Fanuc TP program (LS listing): FM152932.ls

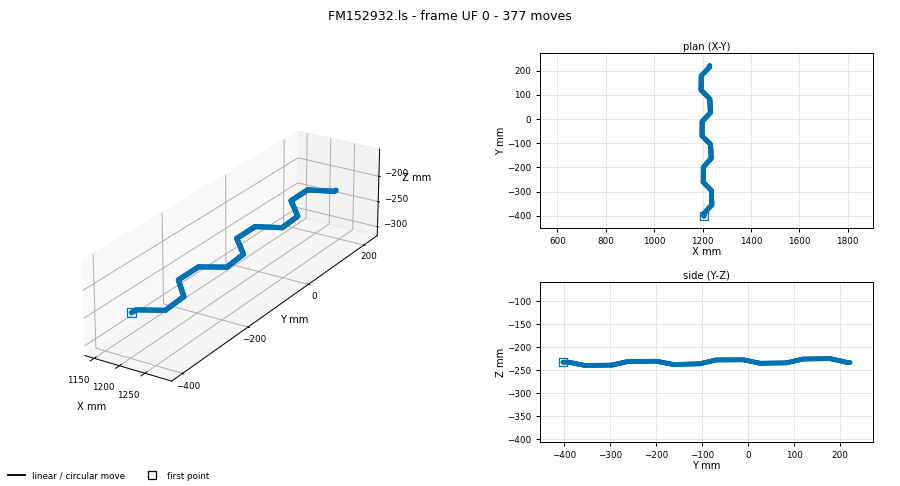
[picture p0: tool path of FM152932.ls in frame UF 0, 377 of 377 moves have a stored position in this frame; points joined in program order, loops and branches not executed]
/PROG  FM152932
/ATTR
OWNER		= MNEDITOR;
COMMENT		= "Auto FANUC move";
PROG_SIZE	= 0;
CREATE		= DATE 26-05-06  TIME 15:29:32;
MODIFIED	= DATE 26-05-06  TIME 15:29:32;
FILE_NAME	= ;
VERSION		= 0;
LINE_COUNT	= 382;
MEMORY_SIZE	= 0;
PROTECT		= READ_WRITE;
TCD:  STACK_SIZE	= 0,
      TASK_PRIORITY	= 50,
      TIME_SLICE	= 0,
      BUSY_LAMP_OFF	= 0,
      ABORT_REQUEST	= 0,
      PAUSE_REQUEST	= 0;
DEFAULT_GROUP	= 1,*,*,*,*;
CONTROL_CODE	= 00000000 00000000;
/MN
   1:  UFRAME_NUM=0 ;
   2:  UTOOL_NUM=1 ;
   3:  R[93]=10 ;
   4:  L P[1] 7mm/sec FINE ;
   5:  L P[2] 7mm/sec CNT50 ;
   6:  L P[3] 7mm/sec CNT50 ;
   7:  L P[4] 7mm/sec CNT50 ;
   8:  L P[5] 7mm/sec CNT50 ;
   9:  L P[6] 7mm/sec CNT50 ;
  10:  L P[7] 7mm/sec CNT50 ;
  11:  L P[8] 7mm/sec CNT50 ;
  12:  L P[9] 7mm/sec CNT50 ;
  13:  L P[10] 7mm/sec CNT50 ;
  14:  L P[11] 7mm/sec CNT50 ;
  15:  L P[12] 7mm/sec CNT50 ;
  16:  L P[13] 7mm/sec CNT50 ;
  17:  L P[14] 7mm/sec CNT50 ;
  18:  L P[15] 7mm/sec CNT50 ;
  19:  L P[16] 7mm/sec CNT50 ;
  20:  L P[17] 7mm/sec CNT50 ;
  21:  L P[18] 7mm/sec CNT50 ;
  22:  L P[19] 7mm/sec CNT50 ;
  23:  L P[20] 7mm/sec CNT50 ;
  24:  L P[21] 7mm/sec CNT50 ;
  25:  L P[22] 7mm/sec CNT50 ;
  26:  L P[23] 7mm/sec CNT50 ;
  27:  L P[24] 7mm/sec CNT50 ;
  28:  L P[25] 7mm/sec CNT50 ;
  29:  L P[26] 7mm/sec CNT50 ;
  30:  L P[27] 7mm/sec CNT50 ;
  31:  L P[28] 7mm/sec CNT50 ;
  32:  L P[29] 7mm/sec CNT50 ;
  33:  L P[30] 7mm/sec CNT50 ;
  34:  L P[31] 7mm/sec CNT50 ;
  35:  L P[32] 7mm/sec CNT50 ;
  36:  L P[33] 7mm/sec CNT50 ;
  37:  L P[34] 7mm/sec CNT50 ;
  38:  L P[35] 7mm/sec CNT50 ;
  39:  L P[36] 7mm/sec CNT50 ;
  40:  L P[37] 7mm/sec CNT50 ;
  41:  L P[38] 7mm/sec CNT50 ;
  42:  L P[39] 7mm/sec CNT50 ;
  43:  L P[40] 7mm/sec CNT50 ;
  44:  L P[41] 7mm/sec CNT50 ;
  45:  L P[42] 7mm/sec CNT50 ;
  46:  L P[43] 7mm/sec CNT50 ;
  47:  L P[44] 7mm/sec CNT50 ;
  48:  L P[45] 7mm/sec CNT50 ;
  49:  L P[46] 7mm/sec CNT50 ;
  50:  L P[47] 7mm/sec CNT50 ;
  51:  L P[48] 7mm/sec CNT50 ;
  52:  L P[49] 7mm/sec CNT50 ;
  53:  L P[50] 7mm/sec CNT50 ;
  54:  L P[51] 7mm/sec CNT50 ;
  55:  L P[52] 7mm/sec CNT50 ;
  56:  L P[53] 7mm/sec CNT50 ;
  57:  L P[54] 7mm/sec CNT50 ;
  58:  L P[55] 7mm/sec CNT50 ;
  59:  L P[56] 7mm/sec CNT50 ;
  60:  L P[57] 7mm/sec CNT50 ;
  61:  L P[58] 7mm/sec CNT50 ;
  62:  L P[59] 7mm/sec CNT50 ;
  63:  L P[60] 7mm/sec CNT50 ;
  64:  L P[61] 7mm/sec CNT50 ;
  65:  L P[62] 7mm/sec CNT50 ;
  66:  L P[63] 7mm/sec CNT50 ;
  67:  L P[64] 7mm/sec CNT50 ;
  68:  L P[65] 7mm/sec CNT50 ;
  69:  L P[66] 7mm/sec CNT50 ;
  70:  L P[67] 7mm/sec CNT50 ;
  71:  L P[68] 7mm/sec CNT50 ;
  72:  L P[69] 7mm/sec CNT50 ;
  73:  L P[70] 7mm/sec CNT50 ;
  74:  L P[71] 7mm/sec CNT50 ;
  75:  L P[72] 7mm/sec CNT50 ;
  76:  L P[73] 7mm/sec CNT50 ;
  77:  L P[74] 7mm/sec CNT50 ;
  78:  L P[75] 7mm/sec CNT50 ;
  79:  L P[76] 7mm/sec CNT50 ;
  80:  L P[77] 7mm/sec CNT50 ;
  81:  L P[78] 7mm/sec CNT50 ;
  82:  L P[79] 7mm/sec CNT50 ;
  83:  L P[80] 7mm/sec CNT50 ;
  84:  L P[81] 7mm/sec CNT50 ;
  85:  L P[82] 7mm/sec CNT50 ;
  86:  L P[83] 7mm/sec CNT50 ;
  87:  L P[84] 7mm/sec CNT50 ;
  88:  L P[85] 7mm/sec CNT50 ;
  89:  L P[86] 7mm/sec CNT50 ;
  90:  L P[87] 7mm/sec CNT50 ;
  91:  L P[88] 7mm/sec CNT50 ;
  92:  L P[89] 7mm/sec CNT50 ;
  93:  L P[90] 7mm/sec CNT50 ;
  94:  L P[91] 7mm/sec CNT50 ;
  95:  L P[92] 7mm/sec CNT50 ;
  96:  L P[93] 7mm/sec CNT50 ;
  97:  L P[94] 7mm/sec CNT50 ;
  98:  L P[95] 7mm/sec CNT50 ;
  99:  L P[96] 7mm/sec CNT50 ;
 100:  L P[97] 7mm/sec CNT50 ;
 101:  L P[98] 7mm/sec CNT50 ;
 102:  L P[99] 7mm/sec CNT50 ;
 103:  L P[100] 7mm/sec CNT50 ;
 104:  L P[101] 7mm/sec CNT50 ;
 105:  L P[102] 7mm/sec CNT50 ;
 106:  L P[103] 7mm/sec CNT50 ;
 107:  L P[104] 7mm/sec CNT50 ;
 108:  L P[105] 7mm/sec CNT50 ;
 109:  L P[106] 7mm/sec CNT50 ;
 110:  L P[107] 7mm/sec CNT50 ;
 111:  L P[108] 7mm/sec CNT50 ;
 112:  L P[109] 7mm/sec CNT50 ;
 113:  L P[110] 7mm/sec CNT50 ;
 114:  L P[111] 7mm/sec CNT50 ;
 115:  L P[112] 7mm/sec CNT50 ;
 116:  L P[113] 7mm/sec CNT50 ;
 117:  L P[114] 7mm/sec CNT50 ;
 118:  L P[115] 7mm/sec CNT50 ;
 119:  L P[116] 7mm/sec CNT50 ;
 120:  L P[117] 7mm/sec CNT50 ;
 121:  L P[118] 7mm/sec CNT50 ;
 122:  L P[119] 7mm/sec CNT50 ;
 123:  L P[120] 7mm/sec CNT50 ;
 124:  L P[121] 7mm/sec CNT50 ;
 125:  L P[122] 7mm/sec CNT50 ;
 126:  L P[123] 7mm/sec CNT50 ;
 127:  L P[124] 7mm/sec CNT50 ;
 128:  L P[125] 7mm/sec CNT50 ;
 129:  L P[126] 7mm/sec CNT50 ;
 130:  L P[127] 7mm/sec CNT50 ;
 131:  L P[128] 7mm/sec CNT50 ;
 132:  L P[129] 7mm/sec CNT50 ;
 133:  L P[130] 7mm/sec CNT50 ;
 134:  L P[131] 7mm/sec CNT50 ;
 135:  L P[132] 7mm/sec CNT50 ;
 136:  L P[133] 7mm/sec CNT50 ;
 137:  L P[134] 7mm/sec CNT50 ;
 138:  L P[135] 7mm/sec CNT50 ;
 139:  L P[136] 7mm/sec CNT50 ;
 140:  L P[137] 7mm/sec CNT50 ;
 141:  L P[138] 7mm/sec CNT50 ;
 142:  L P[139] 7mm/sec CNT50 ;
 143:  L P[140] 7mm/sec CNT50 ;
 144:  L P[141] 7mm/sec CNT50 ;
 145:  L P[142] 7mm/sec CNT50 ;
 146:  L P[143] 7mm/sec CNT50 ;
 147:  L P[144] 7mm/sec CNT50 ;
 148:  L P[145] 7mm/sec CNT50 ;
 149:  L P[146] 7mm/sec CNT50 ;
 150:  L P[147] 7mm/sec CNT50 ;
 151:  L P[148] 7mm/sec CNT50 ;
 152:  L P[149] 7mm/sec CNT50 ;
 153:  L P[150] 7mm/sec CNT50 ;
 154:  L P[151] 7mm/sec CNT50 ;
 155:  L P[152] 7mm/sec CNT50 ;
 156:  L P[153] 7mm/sec CNT50 ;
 157:  L P[154] 7mm/sec CNT50 ;
 158:  L P[155] 7mm/sec CNT50 ;
 159:  L P[156] 7mm/sec CNT50 ;
 160:  L P[157] 7mm/sec CNT50 ;
 161:  L P[158] 7mm/sec CNT50 ;
 162:  L P[159] 7mm/sec CNT50 ;
 163:  L P[160] 7mm/sec CNT50 ;
 164:  L P[161] 7mm/sec CNT50 ;
 165:  L P[162] 7mm/sec CNT50 ;
 166:  L P[163] 7mm/sec CNT50 ;
 167:  L P[164] 7mm/sec CNT50 ;
 168:  L P[165] 7mm/sec CNT50 ;
 169:  L P[166] 7mm/sec CNT50 ;
 170:  L P[167] 7mm/sec CNT50 ;
 171:  L P[168] 7mm/sec CNT50 ;
 172:  L P[169] 7mm/sec CNT50 ;
 173:  L P[170] 7mm/sec CNT50 ;
 174:  L P[171] 7mm/sec CNT50 ;
 175:  L P[172] 7mm/sec CNT50 ;
 176:  L P[173] 7mm/sec CNT50 ;
 177:  L P[174] 7mm/sec CNT50 ;
 178:  L P[175] 7mm/sec CNT50 ;
 179:  L P[176] 7mm/sec CNT50 ;
 180:  L P[177] 7mm/sec CNT50 ;
 181:  L P[178] 7mm/sec CNT50 ;
 182:  L P[179] 7mm/sec CNT50 ;
 183:  L P[180] 7mm/sec CNT50 ;
 184:  L P[181] 7mm/sec CNT50 ;
 185:  L P[182] 7mm/sec CNT50 ;
 186:  L P[183] 7mm/sec CNT50 ;
 187:  L P[184] 7mm/sec CNT50 ;
 188:  L P[185] 7mm/sec CNT50 ;
 189:  L P[186] 7mm/sec CNT50 ;
 190:  L P[187] 7mm/sec CNT50 ;
 191:  L P[188] 7mm/sec CNT50 ;
 192:  L P[189] 7mm/sec CNT50 ;
 193:  L P[190] 7mm/sec CNT50 ;
 194:  L P[191] 7mm/sec CNT50 ;
 195:  L P[192] 7mm/sec CNT50 ;
 196:  L P[193] 7mm/sec CNT50 ;
 197:  L P[194] 7mm/sec CNT50 ;
 198:  L P[195] 7mm/sec CNT50 ;
 199:  L P[196] 7mm/sec CNT50 ;
 200:  L P[197] 7mm/sec CNT50 ;
 201:  L P[198] 7mm/sec CNT50 ;
 202:  L P[199] 7mm/sec CNT50 ;
 203:  L P[200] 7mm/sec CNT50 ;
 204:  L P[201] 7mm/sec CNT50 ;
 205:  L P[202] 7mm/sec CNT50 ;
 206:  L P[203] 7mm/sec CNT50 ;
 207:  L P[204] 7mm/sec CNT50 ;
 208:  L P[205] 7mm/sec CNT50 ;
 209:  L P[206] 7mm/sec CNT50 ;
 210:  L P[207] 7mm/sec CNT50 ;
 211:  L P[208] 7mm/sec CNT50 ;
 212:  L P[209] 7mm/sec CNT50 ;
 213:  L P[210] 7mm/sec CNT50 ;
 214:  L P[211] 7mm/sec CNT50 ;
 215:  L P[212] 7mm/sec CNT50 ;
 216:  L P[213] 7mm/sec CNT50 ;
 217:  L P[214] 7mm/sec CNT50 ;
 218:  L P[215] 7mm/sec CNT50 ;
 219:  L P[216] 7mm/sec CNT50 ;
 220:  L P[217] 7mm/sec CNT50 ;
 221:  L P[218] 7mm/sec CNT50 ;
 222:  L P[219] 7mm/sec CNT50 ;
 223:  L P[220] 7mm/sec CNT50 ;
 224:  L P[221] 7mm/sec CNT50 ;
 225:  L P[222] 7mm/sec CNT50 ;
 226:  L P[223] 7mm/sec CNT50 ;
 227:  L P[224] 7mm/sec CNT50 ;
 228:  L P[225] 7mm/sec CNT50 ;
 229:  L P[226] 7mm/sec CNT50 ;
 230:  L P[227] 7mm/sec CNT50 ;
 231:  L P[228] 7mm/sec CNT50 ;
 232:  L P[229] 7mm/sec CNT50 ;
 233:  L P[230] 7mm/sec CNT50 ;
 234:  L P[231] 7mm/sec CNT50 ;
 235:  L P[232] 7mm/sec CNT50 ;
 236:  L P[233] 7mm/sec CNT50 ;
 237:  L P[234] 7mm/sec CNT50 ;
 238:  L P[235] 7mm/sec CNT50 ;
 239:  L P[236] 7mm/sec CNT50 ;
 240:  L P[237] 7mm/sec CNT50 ;
 241:  L P[238] 7mm/sec CNT50 ;
 242:  L P[239] 7mm/sec CNT50 ;
 243:  L P[240] 7mm/sec CNT50 ;
 244:  L P[241] 7mm/sec CNT50 ;
 245:  L P[242] 7mm/sec CNT50 ;
 246:  L P[243] 7mm/sec CNT50 ;
 247:  L P[244] 7mm/sec CNT50 ;
 248:  L P[245] 7mm/sec CNT50 ;
 249:  L P[246] 7mm/sec CNT50 ;
 250:  L P[247] 7mm/sec CNT50 ;
 251:  L P[248] 7mm/sec CNT50 ;
 252:  L P[249] 7mm/sec CNT50 ;
 253:  L P[250] 7mm/sec CNT50 ;
 254:  L P[251] 7mm/sec CNT50 ;
 255:  L P[252] 7mm/sec CNT50 ;
 256:  L P[253] 7mm/sec CNT50 ;
 257:  L P[254] 7mm/sec CNT50 ;
 258:  L P[255] 7mm/sec CNT50 ;
 259:  L P[256] 7mm/sec CNT50 ;
 260:  L P[257] 7mm/sec CNT50 ;
 261:  L P[258] 7mm/sec CNT50 ;
 262:  L P[259] 7mm/sec CNT50 ;
 263:  L P[260] 7mm/sec CNT50 ;
 264:  L P[261] 7mm/sec CNT50 ;
 265:  L P[262] 7mm/sec CNT50 ;
 266:  L P[263] 7mm/sec CNT50 ;
 267:  L P[264] 7mm/sec CNT50 ;
 268:  L P[265] 7mm/sec CNT50 ;
 269:  L P[266] 7mm/sec CNT50 ;
 270:  L P[267] 7mm/sec CNT50 ;
 271:  L P[268] 7mm/sec CNT50 ;
 272:  L P[269] 7mm/sec CNT50 ;
 273:  L P[270] 7mm/sec CNT50 ;
 274:  L P[271] 7mm/sec CNT50 ;
 275:  L P[272] 7mm/sec CNT50 ;
 276:  L P[273] 7mm/sec CNT50 ;
 277:  L P[274] 7mm/sec CNT50 ;
 278:  L P[275] 7mm/sec CNT50 ;
 279:  L P[276] 7mm/sec CNT50 ;
 280:  L P[277] 7mm/sec CNT50 ;
 281:  L P[278] 7mm/sec CNT50 ;
 282:  L P[279] 7mm/sec CNT50 ;
 283:  L P[280] 7mm/sec CNT50 ;
 284:  L P[281] 7mm/sec CNT50 ;
 285:  L P[282] 7mm/sec CNT50 ;
 286:  L P[283] 7mm/sec CNT50 ;
 287:  L P[284] 7mm/sec CNT50 ;
 288:  L P[285] 7mm/sec CNT50 ;
 289:  L P[286] 7mm/sec CNT50 ;
 290:  L P[287] 7mm/sec CNT50 ;
 291:  L P[288] 7mm/sec CNT50 ;
 292:  L P[289] 7mm/sec CNT50 ;
 293:  L P[290] 7mm/sec CNT50 ;
 294:  L P[291] 7mm/sec CNT50 ;
 295:  L P[292] 7mm/sec CNT50 ;
 296:  L P[293] 7mm/sec CNT50 ;
 297:  L P[294] 7mm/sec CNT50 ;
 298:  L P[295] 7mm/sec CNT50 ;
 299:  L P[296] 7mm/sec CNT50 ;
 300:  L P[297] 7mm/sec CNT50 ;
 301:  L P[298] 7mm/sec CNT50 ;
 302:  L P[299] 7mm/sec CNT50 ;
 303:  L P[300] 7mm/sec CNT50 ;
 304:  L P[301] 7mm/sec CNT50 ;
 305:  L P[302] 7mm/sec CNT50 ;
 306:  L P[303] 7mm/sec CNT50 ;
 307:  L P[304] 7mm/sec CNT50 ;
 308:  L P[305] 7mm/sec CNT50 ;
 309:  L P[306] 7mm/sec CNT50 ;
 310:  L P[307] 7mm/sec CNT50 ;
 311:  L P[308] 7mm/sec CNT50 ;
 312:  L P[309] 7mm/sec CNT50 ;
 313:  L P[310] 7mm/sec CNT50 ;
 314:  L P[311] 7mm/sec CNT50 ;
 315:  L P[312] 7mm/sec CNT50 ;
 316:  L P[313] 7mm/sec CNT50 ;
 317:  L P[314] 7mm/sec CNT50 ;
 318:  L P[315] 7mm/sec CNT50 ;
 319:  L P[316] 7mm/sec CNT50 ;
 320:  L P[317] 7mm/sec CNT50 ;
 321:  L P[318] 7mm/sec CNT50 ;
 322:  L P[319] 7mm/sec CNT50 ;
 323:  L P[320] 7mm/sec CNT50 ;
 324:  L P[321] 7mm/sec CNT50 ;
 325:  L P[322] 7mm/sec CNT50 ;
 326:  L P[323] 7mm/sec CNT50 ;
 327:  L P[324] 7mm/sec CNT50 ;
 328:  L P[325] 7mm/sec CNT50 ;
 329:  L P[326] 7mm/sec CNT50 ;
 330:  L P[327] 7mm/sec CNT50 ;
 331:  L P[328] 7mm/sec CNT50 ;
 332:  L P[329] 7mm/sec CNT50 ;
 333:  L P[330] 7mm/sec CNT50 ;
 334:  L P[331] 7mm/sec CNT50 ;
 335:  L P[332] 7mm/sec CNT50 ;
 336:  L P[333] 7mm/sec CNT50 ;
 337:  L P[334] 7mm/sec CNT50 ;
 338:  L P[335] 7mm/sec CNT50 ;
 339:  L P[336] 7mm/sec CNT50 ;
 340:  L P[337] 7mm/sec CNT50 ;
 341:  L P[338] 7mm/sec CNT50 ;
 342:  L P[339] 7mm/sec CNT50 ;
 343:  L P[340] 7mm/sec CNT50 ;
 344:  L P[341] 7mm/sec CNT50 ;
 345:  L P[342] 7mm/sec CNT50 ;
 346:  L P[343] 7mm/sec CNT50 ;
 347:  L P[344] 7mm/sec CNT50 ;
 348:  L P[345] 7mm/sec CNT50 ;
 349:  L P[346] 7mm/sec CNT50 ;
 350:  L P[347] 7mm/sec CNT50 ;
 351:  L P[348] 7mm/sec CNT50 ;
 352:  L P[349] 7mm/sec CNT50 ;
 353:  L P[350] 7mm/sec CNT50 ;
 354:  L P[351] 7mm/sec CNT50 ;
 355:  L P[352] 7mm/sec CNT50 ;
 356:  L P[353] 7mm/sec CNT50 ;
 357:  L P[354] 7mm/sec CNT50 ;
 358:  L P[355] 7mm/sec CNT50 ;
 359:  L P[356] 7mm/sec CNT50 ;
 360:  L P[357] 7mm/sec CNT50 ;
 361:  L P[358] 7mm/sec CNT50 ;
 362:  L P[359] 7mm/sec CNT50 ;
 363:  L P[360] 7mm/sec CNT50 ;
 364:  L P[361] 7mm/sec CNT50 ;
 365:  L P[362] 7mm/sec CNT50 ;
 366:  L P[363] 7mm/sec CNT50 ;
 367:  L P[364] 7mm/sec CNT50 ;
 368:  L P[365] 7mm/sec CNT50 ;
 369:  L P[366] 7mm/sec CNT50 ;
 370:  L P[367] 7mm/sec CNT50 ;
 371:  L P[368] 7mm/sec CNT50 ;
 372:  L P[369] 7mm/sec CNT50 ;
 373:  L P[370] 7mm/sec CNT50 ;
 374:  L P[371] 7mm/sec CNT50 ;
 375:  L P[372] 7mm/sec CNT50 ;
 376:  L P[373] 7mm/sec CNT50 ;
 377:  L P[374] 7mm/sec CNT50 ;
 378:  L P[375] 7mm/sec CNT50 ;
 379:  L P[376] 7mm/sec CNT50 ;
 380:  L P[377] 7mm/sec FINE ;
 381:  R[93]=1 ;
 382:  END ;
/POS
P[1]{
   GP1:
	UF : 0, UT : 1,		CONFIG : 'N U T, 0, 0, 0',
	X = 1205.571  mm,	Y = -402.138  mm,	Z = -232.677  mm,
	W = 0.000 deg,	P = 30.000 deg,	R = 176.726 deg
};
P[2]{
   GP1:
	UF : 0, UT : 1,		CONFIG : 'N U T, 0, 0, 0',
	X = 1205.685  mm,	Y = -400.142  mm,	Z = -232.675  mm,
	W = 0.000 deg,	P = 30.000 deg,	R = 176.726 deg
};
P[3]{
   GP1:
	UF : 0, UT : 1,		CONFIG : 'N U T, 0, 0, 0',
	X = 1205.800  mm,	Y = -398.145  mm,	Z = -232.673  mm,
	W = 0.000 deg,	P = 30.000 deg,	R = 173.381 deg
};
P[4]{
   GP1:
	UF : 0, UT : 1,		CONFIG : 'N U T, 0, 0, 0',
	X = 1205.914  mm,	Y = -396.148  mm,	Z = -232.672  mm,
	W = 0.000 deg,	P = 30.000 deg,	R = 170.036 deg
};
P[5]{
   GP1:
	UF : 0, UT : 1,		CONFIG : 'N U T, 0, 0, 0',
	X = 1206.028  mm,	Y = -394.151  mm,	Z = -232.670  mm,
	W = 0.000 deg,	P = 30.000 deg,	R = 166.691 deg
};
P[6]{
   GP1:
	UF : 0, UT : 1,		CONFIG : 'N U T, 0, 0, 0',
	X = 1206.142  mm,	Y = -392.155  mm,	Z = -232.668  mm,
	W = 0.000 deg,	P = 30.000 deg,	R = 163.345 deg
};
P[7]{
   GP1:
	UF : 0, UT : 1,		CONFIG : 'N U T, 0, 0, 0',
	X = 1206.257  mm,	Y = -390.158  mm,	Z = -232.666  mm,
	W = 0.000 deg,	P = 30.000 deg,	R = 160.000 deg
};
P[8]{
   GP1:
	UF : 0, UT : 1,		CONFIG : 'N U T, 0, 0, 0',
	X = 1206.293  mm,	Y = -389.526  mm,	Z = -232.666  mm,
	W = 0.000 deg,	P = 30.000 deg,	R = 160.000 deg
};
P[9]{
   GP1:
	UF : 0, UT : 1,		CONFIG : 'N U T, 0, 0, 0',
	X = 1207.204  mm,	Y = -388.527  mm,	Z = -232.864  mm,
	W = 0.000 deg,	P = 30.000 deg,	R = 160.000 deg
};
P[10]{
   GP1:
	UF : 0, UT : 1,		CONFIG : 'N U T, 0, 0, 0',
	X = 1208.538  mm,	Y = -387.065  mm,	Z = -233.154  mm,
	W = 0.000 deg,	P = 30.000 deg,	R = 160.000 deg
};
P[11]{
   GP1:
	UF : 0, UT : 1,		CONFIG : 'N U T, 0, 0, 0',
	X = 1209.872  mm,	Y = -385.603  mm,	Z = -233.445  mm,
	W = 0.000 deg,	P = 30.000 deg,	R = 160.000 deg
};
P[12]{
   GP1:
	UF : 0, UT : 1,		CONFIG : 'N U T, 0, 0, 0',
	X = 1211.205  mm,	Y = -384.141  mm,	Z = -233.735  mm,
	W = 0.000 deg,	P = 30.000 deg,	R = 160.000 deg
};
P[13]{
   GP1:
	UF : 0, UT : 1,		CONFIG : 'N U T, 0, 0, 0',
	X = 1212.539  mm,	Y = -382.679  mm,	Z = -234.025  mm,
	W = 0.000 deg,	P = 30.000 deg,	R = 160.000 deg
};
P[14]{
   GP1:
	UF : 0, UT : 1,		CONFIG : 'N U T, 0, 0, 0',
	X = 1213.873  mm,	Y = -381.217  mm,	Z = -234.315  mm,
	W = 0.000 deg,	P = 30.000 deg,	R = 160.000 deg
};
P[15]{
   GP1:
	UF : 0, UT : 1,		CONFIG : 'N U T, 0, 0, 0',
	X = 1215.206  mm,	Y = -379.755  mm,	Z = -234.605  mm,
	W = 0.000 deg,	P = 30.000 deg,	R = 160.000 deg
};
P[16]{
   GP1:
	UF : 0, UT : 1,		CONFIG : 'N U T, 0, 0, 0',
	X = 1216.540  mm,	Y = -378.294  mm,	Z = -234.896  mm,
	W = 0.000 deg,	P = 30.000 deg,	R = 160.000 deg
};
P[17]{
   GP1:
	UF : 0, UT : 1,		CONFIG : 'N U T, 0, 0, 0',
	X = 1217.874  mm,	Y = -376.832  mm,	Z = -235.186  mm,
	W = 0.000 deg,	P = 30.000 deg,	R = 160.000 deg
};
P[18]{
   GP1:
	UF : 0, UT : 1,		CONFIG : 'N U T, 0, 0, 0',
	X = 1219.207  mm,	Y = -375.370  mm,	Z = -235.476  mm,
	W = 0.000 deg,	P = 30.000 deg,	R = 160.000 deg
};
P[19]{
   GP1:
	UF : 0, UT : 1,		CONFIG : 'N U T, 0, 0, 0',
	X = 1220.541  mm,	Y = -373.908  mm,	Z = -235.766  mm,
	W = 0.000 deg,	P = 30.000 deg,	R = 160.000 deg
};
P[20]{
   GP1:
	UF : 0, UT : 1,		CONFIG : 'N U T, 0, 0, 0',
	X = 1221.875  mm,	Y = -372.446  mm,	Z = -236.056  mm,
	W = 0.000 deg,	P = 30.000 deg,	R = 160.000 deg
};
P[21]{
   GP1:
	UF : 0, UT : 1,		CONFIG : 'N U T, 0, 0, 0',
	X = 1223.208  mm,	Y = -370.984  mm,	Z = -236.346  mm,
	W = 0.000 deg,	P = 30.000 deg,	R = 160.000 deg
};
P[22]{
   GP1:
	UF : 0, UT : 1,		CONFIG : 'N U T, 0, 0, 0',
	X = 1224.542  mm,	Y = -369.522  mm,	Z = -236.637  mm,
	W = 0.000 deg,	P = 30.000 deg,	R = 160.000 deg
};
P[23]{
   GP1:
	UF : 0, UT : 1,		CONFIG : 'N U T, 0, 0, 0',
	X = 1225.876  mm,	Y = -368.060  mm,	Z = -236.927  mm,
	W = 0.000 deg,	P = 30.000 deg,	R = 160.000 deg
};
P[24]{
   GP1:
	UF : 0, UT : 1,		CONFIG : 'N U T, 0, 0, 0',
	X = 1227.209  mm,	Y = -366.598  mm,	Z = -237.217  mm,
	W = 0.000 deg,	P = 30.000 deg,	R = 160.000 deg
};
P[25]{
   GP1:
	UF : 0, UT : 1,		CONFIG : 'N U T, 0, 0, 0',
	X = 1228.543  mm,	Y = -365.136  mm,	Z = -237.507  mm,
	W = 0.000 deg,	P = 30.000 deg,	R = 160.000 deg
};
P[26]{
   GP1:
	UF : 0, UT : 1,		CONFIG : 'N U T, 0, 0, 0',
	X = 1229.877  mm,	Y = -363.674  mm,	Z = -237.797  mm,
	W = 0.000 deg,	P = 30.000 deg,	R = 160.000 deg
};
P[27]{
   GP1:
	UF : 0, UT : 1,		CONFIG : 'N U T, 0, 0, 0',
	X = 1231.210  mm,	Y = -362.213  mm,	Z = -238.087  mm,
	W = 0.000 deg,	P = 30.000 deg,	R = 160.000 deg
};
P[28]{
   GP1:
	UF : 0, UT : 1,		CONFIG : 'N U T, 0, 0, 0',
	X = 1232.544  mm,	Y = -360.751  mm,	Z = -238.378  mm,
	W = 0.000 deg,	P = 30.000 deg,	R = 163.000 deg
};
P[29]{
   GP1:
	UF : 0, UT : 1,		CONFIG : 'N U T, 0, 0, 0',
	X = 1233.878  mm,	Y = -359.289  mm,	Z = -238.668  mm,
	W = 0.000 deg,	P = 30.000 deg,	R = 167.389 deg
};
P[30]{
   GP1:
	UF : 0, UT : 1,		CONFIG : 'N U T, 0, 0, 0',
	X = 1235.211  mm,	Y = -357.827  mm,	Z = -238.958  mm,
	W = 0.000 deg,	P = 30.000 deg,	R = 171.777 deg
};
P[31]{
   GP1:
	UF : 0, UT : 1,		CONFIG : 'N U T, 0, 0, 0',
	X = 1236.545  mm,	Y = -356.365  mm,	Z = -239.248  mm,
	W = 0.000 deg,	P = 30.000 deg,	R = 176.166 deg
};
P[32]{
   GP1:
	UF : 0, UT : 1,		CONFIG : 'N U T, 0, 0, 0',
	X = 1237.879  mm,	Y = -354.903  mm,	Z = -239.538  mm,
	W = 0.000 deg,	P = 30.000 deg,	R = -179.446 deg
};
P[33]{
   GP1:
	UF : 0, UT : 1,		CONFIG : 'N U T, 0, 0, 0',
	X = 1238.755  mm,	Y = -353.942  mm,	Z = -239.729  mm,
	W = 0.000 deg,	P = 30.000 deg,	R = -178.058 deg
};
P[34]{
   GP1:
	UF : 0, UT : 1,		CONFIG : 'N U T, 0, 0, 0',
	X = 1238.732  mm,	Y = -353.257  mm,	Z = -239.719  mm,
	W = 0.000 deg,	P = 30.000 deg,	R = -178.058 deg
};
P[35]{
   GP1:
	UF : 0, UT : 1,		CONFIG : 'N U T, 0, 0, 0',
	X = 1238.664  mm,	Y = -351.259  mm,	Z = -239.691  mm,
	W = 0.000 deg,	P = 30.000 deg,	R = -178.058 deg
};
P[36]{
   GP1:
	UF : 0, UT : 1,		CONFIG : 'N U T, 0, 0, 0',
	X = 1238.597  mm,	Y = -349.260  mm,	Z = -239.662  mm,
	W = 0.000 deg,	P = 30.000 deg,	R = -178.058 deg
};
P[37]{
   GP1:
	UF : 0, UT : 1,		CONFIG : 'N U T, 0, 0, 0',
	X = 1238.529  mm,	Y = -347.261  mm,	Z = -239.633  mm,
	W = 0.000 deg,	P = 30.000 deg,	R = -178.058 deg
};
P[38]{
   GP1:
	UF : 0, UT : 1,		CONFIG : 'N U T, 0, 0, 0',
	X = 1238.461  mm,	Y = -345.263  mm,	Z = -239.605  mm,
	W = 0.000 deg,	P = 30.000 deg,	R = -178.058 deg
};
P[39]{
   GP1:
	UF : 0, UT : 1,		CONFIG : 'N U T, 0, 0, 0',
	X = 1238.393  mm,	Y = -343.264  mm,	Z = -239.576  mm,
	W = 0.000 deg,	P = 30.000 deg,	R = -178.058 deg
};
P[40]{
   GP1:
	UF : 0, UT : 1,		CONFIG : 'N U T, 0, 0, 0',
	X = 1238.325  mm,	Y = -341.265  mm,	Z = -239.547  mm,
	W = 0.000 deg,	P = 30.000 deg,	R = -178.058 deg
};
P[41]{
   GP1:
	UF : 0, UT : 1,		CONFIG : 'N U T, 0, 0, 0',
	X = 1238.258  mm,	Y = -339.267  mm,	Z = -239.519  mm,
	W = 0.000 deg,	P = 30.000 deg,	R = -178.058 deg
};
P[42]{
   GP1:
	UF : 0, UT : 1,		CONFIG : 'N U T, 0, 0, 0',
	X = 1238.190  mm,	Y = -337.268  mm,	Z = -239.490  mm,
	W = 0.000 deg,	P = 30.000 deg,	R = -178.058 deg
};
P[43]{
   GP1:
	UF : 0, UT : 1,		CONFIG : 'N U T, 0, 0, 0',
	X = 1238.122  mm,	Y = -335.269  mm,	Z = -239.461  mm,
	W = 0.000 deg,	P = 30.000 deg,	R = -178.058 deg
};
P[44]{
   GP1:
	UF : 0, UT : 1,		CONFIG : 'N U T, 0, 0, 0',
	X = 1238.054  mm,	Y = -333.271  mm,	Z = -239.433  mm,
	W = 0.000 deg,	P = 30.000 deg,	R = -178.058 deg
};
P[45]{
   GP1:
	UF : 0, UT : 1,		CONFIG : 'N U T, 0, 0, 0',
	X = 1237.987  mm,	Y = -331.272  mm,	Z = -239.404  mm,
	W = 0.000 deg,	P = 30.000 deg,	R = -178.058 deg
};
P[46]{
   GP1:
	UF : 0, UT : 1,		CONFIG : 'N U T, 0, 0, 0',
	X = 1237.919  mm,	Y = -329.274  mm,	Z = -239.375  mm,
	W = 0.000 deg,	P = 30.000 deg,	R = -178.058 deg
};
P[47]{
   GP1:
	UF : 0, UT : 1,		CONFIG : 'N U T, 0, 0, 0',
	X = 1237.851  mm,	Y = -327.275  mm,	Z = -239.347  mm,
	W = 0.000 deg,	P = 30.000 deg,	R = -178.058 deg
};
P[48]{
   GP1:
	UF : 0, UT : 1,		CONFIG : 'N U T, 0, 0, 0',
	X = 1237.783  mm,	Y = -325.276  mm,	Z = -239.318  mm,
	W = 0.000 deg,	P = 30.000 deg,	R = -178.058 deg
};
P[49]{
   GP1:
	UF : 0, UT : 1,		CONFIG : 'N U T, 0, 0, 0',
	X = 1237.715  mm,	Y = -323.278  mm,	Z = -239.289  mm,
	W = 0.000 deg,	P = 30.000 deg,	R = -178.058 deg
};
P[50]{
   GP1:
	UF : 0, UT : 1,		CONFIG : 'N U T, 0, 0, 0',
	X = 1237.648  mm,	Y = -321.279  mm,	Z = -239.261  mm,
	W = 0.000 deg,	P = 30.000 deg,	R = -178.058 deg
};
P[51]{
   GP1:
	UF : 0, UT : 1,		CONFIG : 'N U T, 0, 0, 0',
	X = 1237.580  mm,	Y = -319.280  mm,	Z = -239.232  mm,
	W = 0.000 deg,	P = 30.000 deg,	R = -178.058 deg
};
P[52]{
   GP1:
	UF : 0, UT : 1,		CONFIG : 'N U T, 0, 0, 0',
	X = 1237.512  mm,	Y = -317.282  mm,	Z = -239.203  mm,
	W = 0.000 deg,	P = 30.000 deg,	R = -178.058 deg
};
P[53]{
   GP1:
	UF : 0, UT : 1,		CONFIG : 'N U T, 0, 0, 0',
	X = 1237.444  mm,	Y = -315.283  mm,	Z = -239.175  mm,
	W = 0.000 deg,	P = 30.000 deg,	R = -178.058 deg
};
P[54]{
   GP1:
	UF : 0, UT : 1,		CONFIG : 'N U T, 0, 0, 0',
	X = 1237.377  mm,	Y = -313.284  mm,	Z = -239.146  mm,
	W = 0.000 deg,	P = 30.000 deg,	R = -178.058 deg
};
P[55]{
   GP1:
	UF : 0, UT : 1,		CONFIG : 'N U T, 0, 0, 0',
	X = 1237.309  mm,	Y = -311.286  mm,	Z = -239.117  mm,
	W = 0.000 deg,	P = 30.000 deg,	R = -178.058 deg
};
P[56]{
   GP1:
	UF : 0, UT : 1,		CONFIG : 'N U T, 0, 0, 0',
	X = 1237.241  mm,	Y = -309.287  mm,	Z = -239.089  mm,
	W = 0.000 deg,	P = 30.000 deg,	R = -178.058 deg
};
P[57]{
   GP1:
	UF : 0, UT : 1,		CONFIG : 'N U T, 0, 0, 0',
	X = 1237.173  mm,	Y = -307.288  mm,	Z = -239.060  mm,
	W = 0.000 deg,	P = 30.000 deg,	R = -178.058 deg
};
P[58]{
   GP1:
	UF : 0, UT : 1,		CONFIG : 'N U T, 0, 0, 0',
	X = 1237.105  mm,	Y = -305.290  mm,	Z = -239.031  mm,
	W = 0.000 deg,	P = 30.000 deg,	R = -178.058 deg
};
P[59]{
   GP1:
	UF : 0, UT : 1,		CONFIG : 'N U T, 0, 0, 0',
	X = 1237.038  mm,	Y = -303.291  mm,	Z = -239.003  mm,
	W = 0.000 deg,	P = 30.000 deg,	R = -173.209 deg
};
P[60]{
   GP1:
	UF : 0, UT : 1,		CONFIG : 'N U T, 0, 0, 0',
	X = 1236.970  mm,	Y = -301.293  mm,	Z = -238.974  mm,
	W = 0.000 deg,	P = 30.000 deg,	R = -169.598 deg
};
P[61]{
   GP1:
	UF : 0, UT : 1,		CONFIG : 'N U T, 0, 0, 0',
	X = 1236.902  mm,	Y = -299.294  mm,	Z = -238.945  mm,
	W = 0.000 deg,	P = 30.000 deg,	R = -165.986 deg
};
P[62]{
   GP1:
	UF : 0, UT : 1,		CONFIG : 'N U T, 0, 0, 0',
	X = 1236.834  mm,	Y = -297.295  mm,	Z = -238.917  mm,
	W = 0.000 deg,	P = 30.000 deg,	R = -162.374 deg
};
P[63]{
   GP1:
	UF : 0, UT : 1,		CONFIG : 'N U T, 0, 0, 0',
	X = 1236.784  mm,	Y = -295.800  mm,	Z = -238.895  mm,
	W = 0.000 deg,	P = 30.000 deg,	R = -160.000 deg
};
P[64]{
   GP1:
	UF : 0, UT : 1,		CONFIG : 'N U T, 0, 0, 0',
	X = 1236.439  mm,	Y = -295.442  mm,	Z = -238.815  mm,
	W = 0.000 deg,	P = 30.000 deg,	R = -160.000 deg
};
P[65]{
   GP1:
	UF : 0, UT : 1,		CONFIG : 'N U T, 0, 0, 0',
	X = 1235.069  mm,	Y = -294.020  mm,	Z = -238.495  mm,
	W = 0.000 deg,	P = 30.000 deg,	R = -160.000 deg
};
P[66]{
   GP1:
	UF : 0, UT : 1,		CONFIG : 'N U T, 0, 0, 0',
	X = 1233.699  mm,	Y = -292.598  mm,	Z = -238.174  mm,
	W = 0.000 deg,	P = 30.000 deg,	R = -160.000 deg
};
P[67]{
   GP1:
	UF : 0, UT : 1,		CONFIG : 'N U T, 0, 0, 0',
	X = 1232.330  mm,	Y = -291.176  mm,	Z = -237.854  mm,
	W = 0.000 deg,	P = 30.000 deg,	R = -160.000 deg
};
P[68]{
   GP1:
	UF : 0, UT : 1,		CONFIG : 'N U T, 0, 0, 0',
	X = 1230.960  mm,	Y = -289.754  mm,	Z = -237.534  mm,
	W = 0.000 deg,	P = 30.000 deg,	R = -160.000 deg
};
P[69]{
   GP1:
	UF : 0, UT : 1,		CONFIG : 'N U T, 0, 0, 0',
	X = 1229.591  mm,	Y = -288.333  mm,	Z = -237.214  mm,
	W = 0.000 deg,	P = 30.000 deg,	R = -160.000 deg
};
P[70]{
   GP1:
	UF : 0, UT : 1,		CONFIG : 'N U T, 0, 0, 0',
	X = 1228.221  mm,	Y = -286.911  mm,	Z = -236.894  mm,
	W = 0.000 deg,	P = 30.000 deg,	R = -160.000 deg
};
P[71]{
   GP1:
	UF : 0, UT : 1,		CONFIG : 'N U T, 0, 0, 0',
	X = 1226.851  mm,	Y = -285.489  mm,	Z = -236.573  mm,
	W = 0.000 deg,	P = 30.000 deg,	R = -160.000 deg
};
P[72]{
   GP1:
	UF : 0, UT : 1,		CONFIG : 'N U T, 0, 0, 0',
	X = 1225.482  mm,	Y = -284.067  mm,	Z = -236.253  mm,
	W = 0.000 deg,	P = 30.000 deg,	R = -160.000 deg
};
P[73]{
   GP1:
	UF : 0, UT : 1,		CONFIG : 'N U T, 0, 0, 0',
	X = 1224.112  mm,	Y = -282.645  mm,	Z = -235.933  mm,
	W = 0.000 deg,	P = 30.000 deg,	R = -160.000 deg
};
P[74]{
   GP1:
	UF : 0, UT : 1,		CONFIG : 'N U T, 0, 0, 0',
	X = 1222.743  mm,	Y = -281.223  mm,	Z = -235.613  mm,
	W = 0.000 deg,	P = 30.000 deg,	R = -160.000 deg
};
P[75]{
   GP1:
	UF : 0, UT : 1,		CONFIG : 'N U T, 0, 0, 0',
	X = 1221.373  mm,	Y = -279.802  mm,	Z = -235.293  mm,
	W = 0.000 deg,	P = 30.000 deg,	R = -160.000 deg
};
P[76]{
   GP1:
	UF : 0, UT : 1,		CONFIG : 'N U T, 0, 0, 0',
	X = 1220.003  mm,	Y = -278.380  mm,	Z = -234.973  mm,
	W = 0.000 deg,	P = 30.000 deg,	R = -160.000 deg
};
P[77]{
   GP1:
	UF : 0, UT : 1,		CONFIG : 'N U T, 0, 0, 0',
	X = 1218.634  mm,	Y = -276.958  mm,	Z = -234.652  mm,
	W = 0.000 deg,	P = 30.000 deg,	R = -160.000 deg
};
P[78]{
   GP1:
	UF : 0, UT : 1,		CONFIG : 'N U T, 0, 0, 0',
	X = 1217.264  mm,	Y = -275.536  mm,	Z = -234.332  mm,
	W = 0.000 deg,	P = 30.000 deg,	R = -160.000 deg
};
P[79]{
   GP1:
	UF : 0, UT : 1,		CONFIG : 'N U T, 0, 0, 0',
	X = 1215.895  mm,	Y = -274.114  mm,	Z = -234.012  mm,
	W = 0.000 deg,	P = 30.000 deg,	R = -160.000 deg
};
P[80]{
   GP1:
	UF : 0, UT : 1,		CONFIG : 'N U T, 0, 0, 0',
	X = 1214.525  mm,	Y = -272.692  mm,	Z = -233.692  mm,
	W = 0.000 deg,	P = 30.000 deg,	R = -160.000 deg
};
P[81]{
   GP1:
	UF : 0, UT : 1,		CONFIG : 'N U T, 0, 0, 0',
	X = 1213.155  mm,	Y = -271.270  mm,	Z = -233.372  mm,
	W = 0.000 deg,	P = 30.000 deg,	R = -160.000 deg
};
P[82]{
   GP1:
	UF : 0, UT : 1,		CONFIG : 'N U T, 0, 0, 0',
	X = 1211.786  mm,	Y = -269.849  mm,	Z = -233.051  mm,
	W = 0.000 deg,	P = 30.000 deg,	R = -160.000 deg
};
P[83]{
   GP1:
	UF : 0, UT : 1,		CONFIG : 'N U T, 0, 0, 0',
	X = 1210.416  mm,	Y = -268.427  mm,	Z = -232.731  mm,
	W = 0.000 deg,	P = 30.000 deg,	R = -161.028 deg
};
P[84]{
   GP1:
	UF : 0, UT : 1,		CONFIG : 'N U T, 0, 0, 0',
	X = 1209.046  mm,	Y = -267.005  mm,	Z = -232.411  mm,
	W = 0.000 deg,	P = 30.000 deg,	R = -165.112 deg
};
P[85]{
   GP1:
	UF : 0, UT : 1,		CONFIG : 'N U T, 0, 0, 0',
	X = 1207.677  mm,	Y = -265.583  mm,	Z = -232.091  mm,
	W = 0.000 deg,	P = 30.000 deg,	R = -169.195 deg
};
P[86]{
   GP1:
	UF : 0, UT : 1,		CONFIG : 'N U T, 0, 0, 0',
	X = 1206.307  mm,	Y = -264.161  mm,	Z = -231.771  mm,
	W = 0.000 deg,	P = 30.000 deg,	R = -173.279 deg
};
P[87]{
   GP1:
	UF : 0, UT : 1,		CONFIG : 'N U T, 0, 0, 0',
	X = 1204.938  mm,	Y = -262.739  mm,	Z = -231.451  mm,
	W = 0.000 deg,	P = 30.000 deg,	R = -177.362 deg
};
P[88]{
   GP1:
	UF : 0, UT : 1,		CONFIG : 'N U T, 0, 0, 0',
	X = 1203.568  mm,	Y = -261.318  mm,	Z = -231.130  mm,
	W = 0.000 deg,	P = 30.000 deg,	R = 179.583 deg
};
P[89]{
   GP1:
	UF : 0, UT : 1,		CONFIG : 'N U T, 0, 0, 0',
	X = 1202.654  mm,	Y = -260.369  mm,	Z = -230.917  mm,
	W = 0.000 deg,	P = 30.000 deg,	R = 179.583 deg
};
P[90]{
   GP1:
	UF : 0, UT : 1,		CONFIG : 'N U T, 0, 0, 0',
	X = 1202.659  mm,	Y = -259.703  mm,	Z = -230.912  mm,
	W = 0.000 deg,	P = 30.000 deg,	R = 179.583 deg
};
P[91]{
   GP1:
	UF : 0, UT : 1,		CONFIG : 'N U T, 0, 0, 0',
	X = 1202.673  mm,	Y = -257.703  mm,	Z = -230.899  mm,
	W = 0.000 deg,	P = 30.000 deg,	R = 179.583 deg
};
P[92]{
   GP1:
	UF : 0, UT : 1,		CONFIG : 'N U T, 0, 0, 0',
	X = 1202.688  mm,	Y = -255.704  mm,	Z = -230.886  mm,
	W = 0.000 deg,	P = 30.000 deg,	R = 179.583 deg
};
P[93]{
   GP1:
	UF : 0, UT : 1,		CONFIG : 'N U T, 0, 0, 0',
	X = 1202.703  mm,	Y = -253.704  mm,	Z = -230.873  mm,
	W = 0.000 deg,	P = 30.000 deg,	R = 179.583 deg
};
P[94]{
   GP1:
	UF : 0, UT : 1,		CONFIG : 'N U T, 0, 0, 0',
	X = 1202.717  mm,	Y = -251.704  mm,	Z = -230.860  mm,
	W = 0.000 deg,	P = 30.000 deg,	R = 179.583 deg
};
P[95]{
   GP1:
	UF : 0, UT : 1,		CONFIG : 'N U T, 0, 0, 0',
	X = 1202.732  mm,	Y = -249.704  mm,	Z = -230.847  mm,
	W = 0.000 deg,	P = 30.000 deg,	R = 179.583 deg
};
P[96]{
   GP1:
	UF : 0, UT : 1,		CONFIG : 'N U T, 0, 0, 0',
	X = 1202.746  mm,	Y = -247.704  mm,	Z = -230.834  mm,
	W = 0.000 deg,	P = 30.000 deg,	R = 179.583 deg
};
P[97]{
   GP1:
	UF : 0, UT : 1,		CONFIG : 'N U T, 0, 0, 0',
	X = 1202.761  mm,	Y = -245.704  mm,	Z = -230.821  mm,
	W = 0.000 deg,	P = 30.000 deg,	R = 179.583 deg
};
P[98]{
   GP1:
	UF : 0, UT : 1,		CONFIG : 'N U T, 0, 0, 0',
	X = 1202.775  mm,	Y = -243.704  mm,	Z = -230.808  mm,
	W = 0.000 deg,	P = 30.000 deg,	R = 179.583 deg
};
P[99]{
   GP1:
	UF : 0, UT : 1,		CONFIG : 'N U T, 0, 0, 0',
	X = 1202.790  mm,	Y = -241.704  mm,	Z = -230.795  mm,
	W = 0.000 deg,	P = 30.000 deg,	R = 179.583 deg
};
P[100]{
   GP1:
	UF : 0, UT : 1,		CONFIG : 'N U T, 0, 0, 0',
	X = 1202.805  mm,	Y = -239.704  mm,	Z = -230.781  mm,
	W = 0.000 deg,	P = 30.000 deg,	R = 179.583 deg
};
P[101]{
   GP1:
	UF : 0, UT : 1,		CONFIG : 'N U T, 0, 0, 0',
	X = 1202.819  mm,	Y = -237.704  mm,	Z = -230.768  mm,
	W = 0.000 deg,	P = 30.000 deg,	R = 179.583 deg
};
P[102]{
   GP1:
	UF : 0, UT : 1,		CONFIG : 'N U T, 0, 0, 0',
	X = 1202.834  mm,	Y = -235.705  mm,	Z = -230.755  mm,
	W = 0.000 deg,	P = 30.000 deg,	R = 179.583 deg
};
P[103]{
   GP1:
	UF : 0, UT : 1,		CONFIG : 'N U T, 0, 0, 0',
	X = 1202.848  mm,	Y = -233.705  mm,	Z = -230.742  mm,
	W = 0.000 deg,	P = 30.000 deg,	R = 179.583 deg
};
P[104]{
   GP1:
	UF : 0, UT : 1,		CONFIG : 'N U T, 0, 0, 0',
	X = 1202.863  mm,	Y = -231.705  mm,	Z = -230.729  mm,
	W = 0.000 deg,	P = 30.000 deg,	R = 179.583 deg
};
P[105]{
   GP1:
	UF : 0, UT : 1,		CONFIG : 'N U T, 0, 0, 0',
	X = 1202.877  mm,	Y = -229.705  mm,	Z = -230.716  mm,
	W = 0.000 deg,	P = 30.000 deg,	R = 179.583 deg
};
P[106]{
   GP1:
	UF : 0, UT : 1,		CONFIG : 'N U T, 0, 0, 0',
	X = 1202.892  mm,	Y = -227.705  mm,	Z = -230.703  mm,
	W = 0.000 deg,	P = 30.000 deg,	R = 179.583 deg
};
P[107]{
   GP1:
	UF : 0, UT : 1,		CONFIG : 'N U T, 0, 0, 0',
	X = 1202.907  mm,	Y = -225.705  mm,	Z = -230.690  mm,
	W = 0.000 deg,	P = 30.000 deg,	R = 179.583 deg
};
P[108]{
   GP1:
	UF : 0, UT : 1,		CONFIG : 'N U T, 0, 0, 0',
	X = 1202.921  mm,	Y = -223.705  mm,	Z = -230.677  mm,
	W = 0.000 deg,	P = 30.000 deg,	R = 179.583 deg
};
P[109]{
   GP1:
	UF : 0, UT : 1,		CONFIG : 'N U T, 0, 0, 0',
	X = 1202.936  mm,	Y = -221.705  mm,	Z = -230.664  mm,
	W = 0.000 deg,	P = 30.000 deg,	R = 179.583 deg
};
P[110]{
   GP1:
	UF : 0, UT : 1,		CONFIG : 'N U T, 0, 0, 0',
	X = 1202.950  mm,	Y = -219.705  mm,	Z = -230.650  mm,
	W = 0.000 deg,	P = 30.000 deg,	R = 179.583 deg
};
P[111]{
   GP1:
	UF : 0, UT : 1,		CONFIG : 'N U T, 0, 0, 0',
	X = 1202.965  mm,	Y = -217.705  mm,	Z = -230.637  mm,
	W = 0.000 deg,	P = 30.000 deg,	R = 179.583 deg
};
P[112]{
   GP1:
	UF : 0, UT : 1,		CONFIG : 'N U T, 0, 0, 0',
	X = 1202.979  mm,	Y = -215.705  mm,	Z = -230.624  mm,
	W = 0.000 deg,	P = 30.000 deg,	R = 179.583 deg
};
P[113]{
   GP1:
	UF : 0, UT : 1,		CONFIG : 'N U T, 0, 0, 0',
	X = 1202.994  mm,	Y = -213.706  mm,	Z = -230.611  mm,
	W = 0.000 deg,	P = 30.000 deg,	R = 179.583 deg
};
P[114]{
   GP1:
	UF : 0, UT : 1,		CONFIG : 'N U T, 0, 0, 0',
	X = 1203.009  mm,	Y = -211.706  mm,	Z = -230.598  mm,
	W = 0.000 deg,	P = 30.000 deg,	R = 179.583 deg
};
P[115]{
   GP1:
	UF : 0, UT : 1,		CONFIG : 'N U T, 0, 0, 0',
	X = 1203.023  mm,	Y = -209.706  mm,	Z = -230.585  mm,
	W = 0.000 deg,	P = 30.000 deg,	R = 179.583 deg
};
P[116]{
   GP1:
	UF : 0, UT : 1,		CONFIG : 'N U T, 0, 0, 0',
	X = 1203.038  mm,	Y = -207.706  mm,	Z = -230.572  mm,
	W = 0.000 deg,	P = 30.000 deg,	R = 174.363 deg
};
P[117]{
   GP1:
	UF : 0, UT : 1,		CONFIG : 'N U T, 0, 0, 0',
	X = 1203.052  mm,	Y = -205.706  mm,	Z = -230.559  mm,
	W = 0.000 deg,	P = 30.000 deg,	R = 170.446 deg
};
P[118]{
   GP1:
	UF : 0, UT : 1,		CONFIG : 'N U T, 0, 0, 0',
	X = 1203.067  mm,	Y = -203.706  mm,	Z = -230.546  mm,
	W = 0.000 deg,	P = 30.000 deg,	R = 166.530 deg
};
P[119]{
   GP1:
	UF : 0, UT : 1,		CONFIG : 'N U T, 0, 0, 0',
	X = 1203.081  mm,	Y = -201.706  mm,	Z = -230.533  mm,
	W = 0.000 deg,	P = 30.000 deg,	R = 162.613 deg
};
P[120]{
   GP1:
	UF : 0, UT : 1,		CONFIG : 'N U T, 0, 0, 0',
	X = 1203.096  mm,	Y = -199.706  mm,	Z = -230.520  mm,
	W = 0.000 deg,	P = 30.000 deg,	R = 160.000 deg
};
P[121]{
   GP1:
	UF : 0, UT : 1,		CONFIG : 'N U T, 0, 0, 0',
	X = 1203.097  mm,	Y = -199.573  mm,	Z = -230.519  mm,
	W = 0.000 deg,	P = 30.000 deg,	R = 160.000 deg
};
P[122]{
   GP1:
	UF : 0, UT : 1,		CONFIG : 'N U T, 0, 0, 0',
	X = 1204.313  mm,	Y = -198.180  mm,	Z = -230.780  mm,
	W = 0.000 deg,	P = 30.000 deg,	R = 160.000 deg
};
P[123]{
   GP1:
	UF : 0, UT : 1,		CONFIG : 'N U T, 0, 0, 0',
	X = 1205.615  mm,	Y = -196.688  mm,	Z = -231.059  mm,
	W = 0.000 deg,	P = 30.000 deg,	R = 160.000 deg
};
P[124]{
   GP1:
	UF : 0, UT : 1,		CONFIG : 'N U T, 0, 0, 0',
	X = 1206.917  mm,	Y = -195.196  mm,	Z = -231.339  mm,
	W = 0.000 deg,	P = 30.000 deg,	R = 160.000 deg
};
P[125]{
   GP1:
	UF : 0, UT : 1,		CONFIG : 'N U T, 0, 0, 0',
	X = 1208.219  mm,	Y = -193.704  mm,	Z = -231.619  mm,
	W = 0.000 deg,	P = 30.000 deg,	R = 160.000 deg
};
P[126]{
   GP1:
	UF : 0, UT : 1,		CONFIG : 'N U T, 0, 0, 0',
	X = 1209.521  mm,	Y = -192.212  mm,	Z = -231.898  mm,
	W = 0.000 deg,	P = 30.000 deg,	R = 160.000 deg
};
P[127]{
   GP1:
	UF : 0, UT : 1,		CONFIG : 'N U T, 0, 0, 0',
	X = 1210.823  mm,	Y = -190.720  mm,	Z = -232.178  mm,
	W = 0.000 deg,	P = 30.000 deg,	R = 160.000 deg
};
P[128]{
   GP1:
	UF : 0, UT : 1,		CONFIG : 'N U T, 0, 0, 0',
	X = 1212.125  mm,	Y = -189.228  mm,	Z = -232.458  mm,
	W = 0.000 deg,	P = 30.000 deg,	R = 160.000 deg
};
P[129]{
   GP1:
	UF : 0, UT : 1,		CONFIG : 'N U T, 0, 0, 0',
	X = 1213.427  mm,	Y = -187.736  mm,	Z = -232.737  mm,
	W = 0.000 deg,	P = 30.000 deg,	R = 160.000 deg
};
P[130]{
   GP1:
	UF : 0, UT : 1,		CONFIG : 'N U T, 0, 0, 0',
	X = 1214.730  mm,	Y = -186.244  mm,	Z = -233.017  mm,
	W = 0.000 deg,	P = 30.000 deg,	R = 160.000 deg
};
P[131]{
   GP1:
	UF : 0, UT : 1,		CONFIG : 'N U T, 0, 0, 0',
	X = 1216.032  mm,	Y = -184.752  mm,	Z = -233.296  mm,
	W = 0.000 deg,	P = 30.000 deg,	R = 160.000 deg
};
P[132]{
   GP1:
	UF : 0, UT : 1,		CONFIG : 'N U T, 0, 0, 0',
	X = 1217.334  mm,	Y = -183.260  mm,	Z = -233.576  mm,
	W = 0.000 deg,	P = 30.000 deg,	R = 160.000 deg
};
P[133]{
   GP1:
	UF : 0, UT : 1,		CONFIG : 'N U T, 0, 0, 0',
	X = 1218.636  mm,	Y = -181.768  mm,	Z = -233.856  mm,
	W = 0.000 deg,	P = 30.000 deg,	R = 160.000 deg
};
P[134]{
   GP1:
	UF : 0, UT : 1,		CONFIG : 'N U T, 0, 0, 0',
	X = 1219.938  mm,	Y = -180.276  mm,	Z = -234.135  mm,
	W = 0.000 deg,	P = 30.000 deg,	R = 160.000 deg
};
P[135]{
   GP1:
	UF : 0, UT : 1,		CONFIG : 'N U T, 0, 0, 0',
	X = 1221.240  mm,	Y = -178.784  mm,	Z = -234.415  mm,
	W = 0.000 deg,	P = 30.000 deg,	R = 160.000 deg
};
P[136]{
   GP1:
	UF : 0, UT : 1,		CONFIG : 'N U T, 0, 0, 0',
	X = 1222.542  mm,	Y = -177.291  mm,	Z = -234.695  mm,
	W = 0.000 deg,	P = 30.000 deg,	R = 160.000 deg
};
P[137]{
   GP1:
	UF : 0, UT : 1,		CONFIG : 'N U T, 0, 0, 0',
	X = 1223.844  mm,	Y = -175.799  mm,	Z = -234.974  mm,
	W = 0.000 deg,	P = 30.000 deg,	R = 160.000 deg
};
P[138]{
   GP1:
	UF : 0, UT : 1,		CONFIG : 'N U T, 0, 0, 0',
	X = 1225.147  mm,	Y = -174.307  mm,	Z = -235.254  mm,
	W = 0.000 deg,	P = 30.000 deg,	R = 160.000 deg
};
P[139]{
   GP1:
	UF : 0, UT : 1,		CONFIG : 'N U T, 0, 0, 0',
	X = 1226.449  mm,	Y = -172.815  mm,	Z = -235.533  mm,
	W = 0.000 deg,	P = 30.000 deg,	R = 160.000 deg
};
P[140]{
   GP1:
	UF : 0, UT : 1,		CONFIG : 'N U T, 0, 0, 0',
	X = 1227.751  mm,	Y = -171.323  mm,	Z = -235.813  mm,
	W = 0.000 deg,	P = 30.000 deg,	R = 160.000 deg
};
P[141]{
   GP1:
	UF : 0, UT : 1,		CONFIG : 'N U T, 0, 0, 0',
	X = 1229.053  mm,	Y = -169.831  mm,	Z = -236.093  mm,
	W = 0.000 deg,	P = 30.000 deg,	R = 160.000 deg
};
P[142]{
   GP1:
	UF : 0, UT : 1,		CONFIG : 'N U T, 0, 0, 0',
	X = 1230.355  mm,	Y = -168.339  mm,	Z = -236.372  mm,
	W = 0.000 deg,	P = 30.000 deg,	R = 164.192 deg
};
P[143]{
   GP1:
	UF : 0, UT : 1,		CONFIG : 'N U T, 0, 0, 0',
	X = 1231.657  mm,	Y = -166.847  mm,	Z = -236.652  mm,
	W = 0.000 deg,	P = 30.000 deg,	R = 168.682 deg
};
P[144]{
   GP1:
	UF : 0, UT : 1,		CONFIG : 'N U T, 0, 0, 0',
	X = 1232.959  mm,	Y = -165.355  mm,	Z = -236.932  mm,
	W = 0.000 deg,	P = 30.000 deg,	R = 173.172 deg
};
P[145]{
   GP1:
	UF : 0, UT : 1,		CONFIG : 'N U T, 0, 0, 0',
	X = 1234.261  mm,	Y = -163.863  mm,	Z = -237.211  mm,
	W = 0.000 deg,	P = 30.000 deg,	R = 177.662 deg
};
P[146]{
   GP1:
	UF : 0, UT : 1,		CONFIG : 'N U T, 0, 0, 0',
	X = 1235.564  mm,	Y = -162.371  mm,	Z = -237.491  mm,
	W = 0.000 deg,	P = 30.000 deg,	R = -177.848 deg
};
P[147]{
   GP1:
	UF : 0, UT : 1,		CONFIG : 'N U T, 0, 0, 0',
	X = 1235.858  mm,	Y = -162.033  mm,	Z = -237.554  mm,
	W = 0.000 deg,	P = 30.000 deg,	R = -177.550 deg
};
P[148]{
   GP1:
	UF : 0, UT : 1,		CONFIG : 'N U T, 0, 0, 0',
	X = 1235.792  mm,	Y = -160.487  mm,	Z = -237.514  mm,
	W = 0.000 deg,	P = 30.000 deg,	R = -177.550 deg
};
P[149]{
   GP1:
	UF : 0, UT : 1,		CONFIG : 'N U T, 0, 0, 0',
	X = 1235.706  mm,	Y = -158.490  mm,	Z = -237.462  mm,
	W = 0.000 deg,	P = 30.000 deg,	R = -177.550 deg
};
P[150]{
   GP1:
	UF : 0, UT : 1,		CONFIG : 'N U T, 0, 0, 0',
	X = 1235.621  mm,	Y = -156.492  mm,	Z = -237.411  mm,
	W = 0.000 deg,	P = 30.000 deg,	R = -177.550 deg
};
P[151]{
   GP1:
	UF : 0, UT : 1,		CONFIG : 'N U T, 0, 0, 0',
	X = 1235.535  mm,	Y = -154.495  mm,	Z = -237.359  mm,
	W = 0.000 deg,	P = 30.000 deg,	R = -177.550 deg
};
P[152]{
   GP1:
	UF : 0, UT : 1,		CONFIG : 'N U T, 0, 0, 0',
	X = 1235.450  mm,	Y = -152.497  mm,	Z = -237.307  mm,
	W = 0.000 deg,	P = 30.000 deg,	R = -177.550 deg
};
P[153]{
   GP1:
	UF : 0, UT : 1,		CONFIG : 'N U T, 0, 0, 0',
	X = 1235.364  mm,	Y = -150.500  mm,	Z = -237.255  mm,
	W = 0.000 deg,	P = 30.000 deg,	R = -177.550 deg
};
P[154]{
   GP1:
	UF : 0, UT : 1,		CONFIG : 'N U T, 0, 0, 0',
	X = 1235.279  mm,	Y = -148.502  mm,	Z = -237.203  mm,
	W = 0.000 deg,	P = 30.000 deg,	R = -177.550 deg
};
P[155]{
   GP1:
	UF : 0, UT : 1,		CONFIG : 'N U T, 0, 0, 0',
	X = 1235.193  mm,	Y = -146.505  mm,	Z = -237.152  mm,
	W = 0.000 deg,	P = 30.000 deg,	R = -177.550 deg
};
P[156]{
   GP1:
	UF : 0, UT : 1,		CONFIG : 'N U T, 0, 0, 0',
	X = 1235.108  mm,	Y = -144.507  mm,	Z = -237.100  mm,
	W = 0.000 deg,	P = 30.000 deg,	R = -177.550 deg
};
P[157]{
   GP1:
	UF : 0, UT : 1,		CONFIG : 'N U T, 0, 0, 0',
	X = 1235.023  mm,	Y = -142.510  mm,	Z = -237.048  mm,
	W = 0.000 deg,	P = 30.000 deg,	R = -177.550 deg
};
P[158]{
   GP1:
	UF : 0, UT : 1,		CONFIG : 'N U T, 0, 0, 0',
	X = 1234.937  mm,	Y = -140.512  mm,	Z = -236.996  mm,
	W = 0.000 deg,	P = 30.000 deg,	R = -177.550 deg
};
P[159]{
   GP1:
	UF : 0, UT : 1,		CONFIG : 'N U T, 0, 0, 0',
	X = 1234.852  mm,	Y = -138.515  mm,	Z = -236.945  mm,
	W = 0.000 deg,	P = 30.000 deg,	R = -177.550 deg
};
P[160]{
   GP1:
	UF : 0, UT : 1,		CONFIG : 'N U T, 0, 0, 0',
	X = 1234.766  mm,	Y = -136.517  mm,	Z = -236.893  mm,
	W = 0.000 deg,	P = 30.000 deg,	R = -177.550 deg
};
P[161]{
   GP1:
	UF : 0, UT : 1,		CONFIG : 'N U T, 0, 0, 0',
	X = 1234.681  mm,	Y = -134.520  mm,	Z = -236.841  mm,
	W = 0.000 deg,	P = 30.000 deg,	R = -177.550 deg
};
P[162]{
   GP1:
	UF : 0, UT : 1,		CONFIG : 'N U T, 0, 0, 0',
	X = 1234.595  mm,	Y = -132.522  mm,	Z = -236.789  mm,
	W = 0.000 deg,	P = 30.000 deg,	R = -177.550 deg
};
P[163]{
   GP1:
	UF : 0, UT : 1,		CONFIG : 'N U T, 0, 0, 0',
	X = 1234.510  mm,	Y = -130.525  mm,	Z = -236.738  mm,
	W = 0.000 deg,	P = 30.000 deg,	R = -177.550 deg
};
P[164]{
   GP1:
	UF : 0, UT : 1,		CONFIG : 'N U T, 0, 0, 0',
	X = 1234.424  mm,	Y = -128.527  mm,	Z = -236.686  mm,
	W = 0.000 deg,	P = 30.000 deg,	R = -177.550 deg
};
P[165]{
   GP1:
	UF : 0, UT : 1,		CONFIG : 'N U T, 0, 0, 0',
	X = 1234.339  mm,	Y = -126.530  mm,	Z = -236.634  mm,
	W = 0.000 deg,	P = 30.000 deg,	R = -177.550 deg
};
P[166]{
   GP1:
	UF : 0, UT : 1,		CONFIG : 'N U T, 0, 0, 0',
	X = 1234.253  mm,	Y = -124.532  mm,	Z = -236.582  mm,
	W = 0.000 deg,	P = 30.000 deg,	R = -177.550 deg
};
P[167]{
   GP1:
	UF : 0, UT : 1,		CONFIG : 'N U T, 0, 0, 0',
	X = 1234.168  mm,	Y = -122.535  mm,	Z = -236.530  mm,
	W = 0.000 deg,	P = 30.000 deg,	R = -177.550 deg
};
P[168]{
   GP1:
	UF : 0, UT : 1,		CONFIG : 'N U T, 0, 0, 0',
	X = 1234.082  mm,	Y = -120.537  mm,	Z = -236.479  mm,
	W = 0.000 deg,	P = 30.000 deg,	R = -177.550 deg
};
P[169]{
   GP1:
	UF : 0, UT : 1,		CONFIG : 'N U T, 0, 0, 0',
	X = 1233.997  mm,	Y = -118.540  mm,	Z = -236.427  mm,
	W = 0.000 deg,	P = 30.000 deg,	R = -177.550 deg
};
P[170]{
   GP1:
	UF : 0, UT : 1,		CONFIG : 'N U T, 0, 0, 0',
	X = 1233.911  mm,	Y = -116.542  mm,	Z = -236.375  mm,
	W = 0.000 deg,	P = 30.000 deg,	R = -177.550 deg
};
P[171]{
   GP1:
	UF : 0, UT : 1,		CONFIG : 'N U T, 0, 0, 0',
	X = 1233.826  mm,	Y = -114.545  mm,	Z = -236.323  mm,
	W = 0.000 deg,	P = 30.000 deg,	R = -174.833 deg
};
P[172]{
   GP1:
	UF : 0, UT : 1,		CONFIG : 'N U T, 0, 0, 0',
	X = 1233.741  mm,	Y = -112.547  mm,	Z = -236.272  mm,
	W = 0.000 deg,	P = 30.000 deg,	R = -171.323 deg
};
P[173]{
   GP1:
	UF : 0, UT : 1,		CONFIG : 'N U T, 0, 0, 0',
	X = 1233.655  mm,	Y = -110.550  mm,	Z = -236.220  mm,
	W = 0.000 deg,	P = 30.000 deg,	R = -167.813 deg
};
P[174]{
   GP1:
	UF : 0, UT : 1,		CONFIG : 'N U T, 0, 0, 0',
	X = 1233.570  mm,	Y = -108.552  mm,	Z = -236.168  mm,
	W = 0.000 deg,	P = 30.000 deg,	R = -164.303 deg
};
P[175]{
   GP1:
	UF : 0, UT : 1,		CONFIG : 'N U T, 0, 0, 0',
	X = 1233.484  mm,	Y = -106.555  mm,	Z = -236.116  mm,
	W = 0.000 deg,	P = 30.000 deg,	R = -160.793 deg
};
P[176]{
   GP1:
	UF : 0, UT : 1,		CONFIG : 'N U T, 0, 0, 0',
	X = 1233.415  mm,	Y = -104.939  mm,	Z = -236.074  mm,
	W = 0.000 deg,	P = 30.000 deg,	R = -160.000 deg
};
P[177]{
   GP1:
	UF : 0, UT : 1,		CONFIG : 'N U T, 0, 0, 0',
	X = 1233.147  mm,	Y = -104.674  mm,	Z = -236.011  mm,
	W = 0.000 deg,	P = 30.000 deg,	R = -160.000 deg
};
P[178]{
   GP1:
	UF : 0, UT : 1,		CONFIG : 'N U T, 0, 0, 0',
	X = 1231.748  mm,	Y = -103.284  mm,	Z = -235.680  mm,
	W = 0.000 deg,	P = 30.000 deg,	R = -160.000 deg
};
P[179]{
   GP1:
	UF : 0, UT : 1,		CONFIG : 'N U T, 0, 0, 0',
	X = 1230.348  mm,	Y = -101.894  mm,	Z = -235.349  mm,
	W = 0.000 deg,	P = 30.000 deg,	R = -160.000 deg
};
P[180]{
   GP1:
	UF : 0, UT : 1,		CONFIG : 'N U T, 0, 0, 0',
	X = 1228.948  mm,	Y = -100.504  mm,	Z = -235.019  mm,
	W = 0.000 deg,	P = 30.000 deg,	R = -160.000 deg
};
P[181]{
   GP1:
	UF : 0, UT : 1,		CONFIG : 'N U T, 0, 0, 0',
	X = 1227.548  mm,	Y = -99.115  mm,	Z = -234.688  mm,
	W = 0.000 deg,	P = 30.000 deg,	R = -160.000 deg
};
P[182]{
   GP1:
	UF : 0, UT : 1,		CONFIG : 'N U T, 0, 0, 0',
	X = 1226.149  mm,	Y = -97.725  mm,	Z = -234.357  mm,
	W = 0.000 deg,	P = 30.000 deg,	R = -160.000 deg
};
P[183]{
   GP1:
	UF : 0, UT : 1,		CONFIG : 'N U T, 0, 0, 0',
	X = 1224.749  mm,	Y = -96.335  mm,	Z = -234.026  mm,
	W = 0.000 deg,	P = 30.000 deg,	R = -160.000 deg
};
P[184]{
   GP1:
	UF : 0, UT : 1,		CONFIG : 'N U T, 0, 0, 0',
	X = 1223.349  mm,	Y = -94.946  mm,	Z = -233.695  mm,
	W = 0.000 deg,	P = 30.000 deg,	R = -160.000 deg
};
P[185]{
   GP1:
	UF : 0, UT : 1,		CONFIG : 'N U T, 0, 0, 0',
	X = 1221.950  mm,	Y = -93.556  mm,	Z = -233.364  mm,
	W = 0.000 deg,	P = 30.000 deg,	R = -160.000 deg
};
P[186]{
   GP1:
	UF : 0, UT : 1,		CONFIG : 'N U T, 0, 0, 0',
	X = 1220.550  mm,	Y = -92.166  mm,	Z = -233.033  mm,
	W = 0.000 deg,	P = 30.000 deg,	R = -160.000 deg
};
P[187]{
   GP1:
	UF : 0, UT : 1,		CONFIG : 'N U T, 0, 0, 0',
	X = 1219.150  mm,	Y = -90.776  mm,	Z = -232.703  mm,
	W = 0.000 deg,	P = 30.000 deg,	R = -160.000 deg
};
P[188]{
   GP1:
	UF : 0, UT : 1,		CONFIG : 'N U T, 0, 0, 0',
	X = 1217.750  mm,	Y = -89.387  mm,	Z = -232.372  mm,
	W = 0.000 deg,	P = 30.000 deg,	R = -160.000 deg
};
P[189]{
   GP1:
	UF : 0, UT : 1,		CONFIG : 'N U T, 0, 0, 0',
	X = 1216.351  mm,	Y = -87.997  mm,	Z = -232.041  mm,
	W = 0.000 deg,	P = 30.000 deg,	R = -160.000 deg
};
P[190]{
   GP1:
	UF : 0, UT : 1,		CONFIG : 'N U T, 0, 0, 0',
	X = 1214.951  mm,	Y = -86.607  mm,	Z = -231.710  mm,
	W = 0.000 deg,	P = 30.000 deg,	R = -160.000 deg
};
P[191]{
   GP1:
	UF : 0, UT : 1,		CONFIG : 'N U T, 0, 0, 0',
	X = 1213.551  mm,	Y = -85.217  mm,	Z = -231.379  mm,
	W = 0.000 deg,	P = 30.000 deg,	R = -160.000 deg
};
P[192]{
   GP1:
	UF : 0, UT : 1,		CONFIG : 'N U T, 0, 0, 0',
	X = 1212.152  mm,	Y = -83.828  mm,	Z = -231.048  mm,
	W = 0.000 deg,	P = 30.000 deg,	R = -160.000 deg
};
P[193]{
   GP1:
	UF : 0, UT : 1,		CONFIG : 'N U T, 0, 0, 0',
	X = 1210.752  mm,	Y = -82.438  mm,	Z = -230.717  mm,
	W = 0.000 deg,	P = 30.000 deg,	R = -160.000 deg
};
P[194]{
   GP1:
	UF : 0, UT : 1,		CONFIG : 'N U T, 0, 0, 0',
	X = 1209.352  mm,	Y = -81.048  mm,	Z = -230.386  mm,
	W = 0.000 deg,	P = 30.000 deg,	R = -160.000 deg
};
P[195]{
   GP1:
	UF : 0, UT : 1,		CONFIG : 'N U T, 0, 0, 0',
	X = 1207.953  mm,	Y = -79.659  mm,	Z = -230.056  mm,
	W = 0.000 deg,	P = 30.000 deg,	R = -160.000 deg
};
P[196]{
   GP1:
	UF : 0, UT : 1,		CONFIG : 'N U T, 0, 0, 0',
	X = 1206.553  mm,	Y = -78.269  mm,	Z = -229.725  mm,
	W = 0.000 deg,	P = 30.000 deg,	R = -160.000 deg
};
P[197]{
   GP1:
	UF : 0, UT : 1,		CONFIG : 'N U T, 0, 0, 0',
	X = 1205.153  mm,	Y = -76.879  mm,	Z = -229.394  mm,
	W = 0.000 deg,	P = 30.000 deg,	R = -160.779 deg
};
P[198]{
   GP1:
	UF : 0, UT : 1,		CONFIG : 'N U T, 0, 0, 0',
	X = 1203.753  mm,	Y = -75.489  mm,	Z = -229.063  mm,
	W = 0.000 deg,	P = 30.000 deg,	R = -164.850 deg
};
P[199]{
   GP1:
	UF : 0, UT : 1,		CONFIG : 'N U T, 0, 0, 0',
	X = 1202.354  mm,	Y = -74.100  mm,	Z = -228.732  mm,
	W = 0.000 deg,	P = 30.000 deg,	R = -168.922 deg
};
P[200]{
   GP1:
	UF : 0, UT : 1,		CONFIG : 'N U T, 0, 0, 0',
	X = 1200.954  mm,	Y = -72.710  mm,	Z = -228.401  mm,
	W = 0.000 deg,	P = 30.000 deg,	R = -172.993 deg
};
P[201]{
   GP1:
	UF : 0, UT : 1,		CONFIG : 'N U T, 0, 0, 0',
	X = 1199.554  mm,	Y = -71.320  mm,	Z = -228.070  mm,
	W = 0.000 deg,	P = 30.000 deg,	R = -177.065 deg
};
P[202]{
   GP1:
	UF : 0, UT : 1,		CONFIG : 'N U T, 0, 0, 0',
	X = 1198.155  mm,	Y = -69.930  mm,	Z = -227.740  mm,
	W = 0.000 deg,	P = 30.000 deg,	R = 179.643 deg
};
P[203]{
   GP1:
	UF : 0, UT : 1,		CONFIG : 'N U T, 0, 0, 0',
	X = 1198.028  mm,	Y = -69.804  mm,	Z = -227.710  mm,
	W = 0.000 deg,	P = 30.000 deg,	R = 179.643 deg
};
P[204]{
   GP1:
	UF : 0, UT : 1,		CONFIG : 'N U T, 0, 0, 0',
	X = 1198.039  mm,	Y = -67.986  mm,	Z = -227.701  mm,
	W = 0.000 deg,	P = 30.000 deg,	R = 179.643 deg
};
P[205]{
   GP1:
	UF : 0, UT : 1,		CONFIG : 'N U T, 0, 0, 0',
	X = 1198.051  mm,	Y = -65.986  mm,	Z = -227.692  mm,
	W = 0.000 deg,	P = 30.000 deg,	R = 179.643 deg
};
P[206]{
   GP1:
	UF : 0, UT : 1,		CONFIG : 'N U T, 0, 0, 0',
	X = 1198.064  mm,	Y = -63.986  mm,	Z = -227.682  mm,
	W = 0.000 deg,	P = 30.000 deg,	R = 179.643 deg
};
P[207]{
   GP1:
	UF : 0, UT : 1,		CONFIG : 'N U T, 0, 0, 0',
	X = 1198.076  mm,	Y = -61.986  mm,	Z = -227.673  mm,
	W = 0.000 deg,	P = 30.000 deg,	R = 179.643 deg
};
P[208]{
   GP1:
	UF : 0, UT : 1,		CONFIG : 'N U T, 0, 0, 0',
	X = 1198.089  mm,	Y = -59.986  mm,	Z = -227.664  mm,
	W = 0.000 deg,	P = 30.000 deg,	R = 179.643 deg
};
P[209]{
   GP1:
	UF : 0, UT : 1,		CONFIG : 'N U T, 0, 0, 0',
	X = 1198.101  mm,	Y = -57.986  mm,	Z = -227.654  mm,
	W = 0.000 deg,	P = 30.000 deg,	R = 179.643 deg
};
P[210]{
   GP1:
	UF : 0, UT : 1,		CONFIG : 'N U T, 0, 0, 0',
	X = 1198.114  mm,	Y = -55.986  mm,	Z = -227.645  mm,
	W = 0.000 deg,	P = 30.000 deg,	R = 179.643 deg
};
P[211]{
   GP1:
	UF : 0, UT : 1,		CONFIG : 'N U T, 0, 0, 0',
	X = 1198.126  mm,	Y = -53.986  mm,	Z = -227.636  mm,
	W = 0.000 deg,	P = 30.000 deg,	R = 179.643 deg
};
P[212]{
   GP1:
	UF : 0, UT : 1,		CONFIG : 'N U T, 0, 0, 0',
	X = 1198.139  mm,	Y = -51.986  mm,	Z = -227.626  mm,
	W = 0.000 deg,	P = 30.000 deg,	R = 179.643 deg
};
P[213]{
   GP1:
	UF : 0, UT : 1,		CONFIG : 'N U T, 0, 0, 0',
	X = 1198.151  mm,	Y = -49.986  mm,	Z = -227.617  mm,
	W = 0.000 deg,	P = 30.000 deg,	R = 179.643 deg
};
P[214]{
   GP1:
	UF : 0, UT : 1,		CONFIG : 'N U T, 0, 0, 0',
	X = 1198.164  mm,	Y = -47.986  mm,	Z = -227.608  mm,
	W = 0.000 deg,	P = 30.000 deg,	R = 179.643 deg
};
P[215]{
   GP1:
	UF : 0, UT : 1,		CONFIG : 'N U T, 0, 0, 0',
	X = 1198.176  mm,	Y = -45.987  mm,	Z = -227.598  mm,
	W = 0.000 deg,	P = 30.000 deg,	R = 179.643 deg
};
P[216]{
   GP1:
	UF : 0, UT : 1,		CONFIG : 'N U T, 0, 0, 0',
	X = 1198.189  mm,	Y = -43.987  mm,	Z = -227.589  mm,
	W = 0.000 deg,	P = 30.000 deg,	R = 179.643 deg
};
P[217]{
   GP1:
	UF : 0, UT : 1,		CONFIG : 'N U T, 0, 0, 0',
	X = 1198.201  mm,	Y = -41.987  mm,	Z = -227.580  mm,
	W = 0.000 deg,	P = 30.000 deg,	R = 179.643 deg
};
P[218]{
   GP1:
	UF : 0, UT : 1,		CONFIG : 'N U T, 0, 0, 0',
	X = 1198.213  mm,	Y = -39.987  mm,	Z = -227.570  mm,
	W = 0.000 deg,	P = 30.000 deg,	R = 179.643 deg
};
P[219]{
   GP1:
	UF : 0, UT : 1,		CONFIG : 'N U T, 0, 0, 0',
	X = 1198.226  mm,	Y = -37.987  mm,	Z = -227.561  mm,
	W = 0.000 deg,	P = 30.000 deg,	R = 179.643 deg
};
P[220]{
   GP1:
	UF : 0, UT : 1,		CONFIG : 'N U T, 0, 0, 0',
	X = 1198.238  mm,	Y = -35.987  mm,	Z = -227.552  mm,
	W = 0.000 deg,	P = 30.000 deg,	R = 179.643 deg
};
P[221]{
   GP1:
	UF : 0, UT : 1,		CONFIG : 'N U T, 0, 0, 0',
	X = 1198.251  mm,	Y = -33.987  mm,	Z = -227.542  mm,
	W = 0.000 deg,	P = 30.000 deg,	R = 179.643 deg
};
P[222]{
   GP1:
	UF : 0, UT : 1,		CONFIG : 'N U T, 0, 0, 0',
	X = 1198.263  mm,	Y = -31.987  mm,	Z = -227.533  mm,
	W = 0.000 deg,	P = 30.000 deg,	R = 179.643 deg
};
P[223]{
   GP1:
	UF : 0, UT : 1,		CONFIG : 'N U T, 0, 0, 0',
	X = 1198.276  mm,	Y = -29.987  mm,	Z = -227.524  mm,
	W = 0.000 deg,	P = 30.000 deg,	R = 179.643 deg
};
P[224]{
   GP1:
	UF : 0, UT : 1,		CONFIG : 'N U T, 0, 0, 0',
	X = 1198.288  mm,	Y = -27.987  mm,	Z = -227.514  mm,
	W = 0.000 deg,	P = 30.000 deg,	R = 179.643 deg
};
P[225]{
   GP1:
	UF : 0, UT : 1,		CONFIG : 'N U T, 0, 0, 0',
	X = 1198.301  mm,	Y = -25.987  mm,	Z = -227.505  mm,
	W = 0.000 deg,	P = 30.000 deg,	R = 179.643 deg
};
P[226]{
   GP1:
	UF : 0, UT : 1,		CONFIG : 'N U T, 0, 0, 0',
	X = 1198.313  mm,	Y = -23.987  mm,	Z = -227.496  mm,
	W = 0.000 deg,	P = 30.000 deg,	R = 179.643 deg
};
P[227]{
   GP1:
	UF : 0, UT : 1,		CONFIG : 'N U T, 0, 0, 0',
	X = 1198.326  mm,	Y = -21.987  mm,	Z = -227.487  mm,
	W = 0.000 deg,	P = 30.000 deg,	R = 179.643 deg
};
P[228]{
   GP1:
	UF : 0, UT : 1,		CONFIG : 'N U T, 0, 0, 0',
	X = 1198.338  mm,	Y = -19.987  mm,	Z = -227.477  mm,
	W = 0.000 deg,	P = 30.000 deg,	R = 176.071 deg
};
P[229]{
   GP1:
	UF : 0, UT : 1,		CONFIG : 'N U T, 0, 0, 0',
	X = 1198.351  mm,	Y = -17.987  mm,	Z = -227.468  mm,
	W = 0.000 deg,	P = 30.000 deg,	R = 172.142 deg
};
P[230]{
   GP1:
	UF : 0, UT : 1,		CONFIG : 'N U T, 0, 0, 0',
	X = 1198.363  mm,	Y = -15.987  mm,	Z = -227.459  mm,
	W = 0.000 deg,	P = 30.000 deg,	R = 168.214 deg
};
P[231]{
   GP1:
	UF : 0, UT : 1,		CONFIG : 'N U T, 0, 0, 0',
	X = 1198.376  mm,	Y = -13.988  mm,	Z = -227.449  mm,
	W = 0.000 deg,	P = 30.000 deg,	R = 164.285 deg
};
P[232]{
   GP1:
	UF : 0, UT : 1,		CONFIG : 'N U T, 0, 0, 0',
	X = 1198.388  mm,	Y = -11.988  mm,	Z = -227.440  mm,
	W = 0.000 deg,	P = 30.000 deg,	R = 160.357 deg
};
P[233]{
   GP1:
	UF : 0, UT : 1,		CONFIG : 'N U T, 0, 0, 0',
	X = 1198.400  mm,	Y = -10.138  mm,	Z = -227.431  mm,
	W = 0.000 deg,	P = 30.000 deg,	R = 160.000 deg
};
P[234]{
   GP1:
	UF : 0, UT : 1,		CONFIG : 'N U T, 0, 0, 0',
	X = 1198.501  mm,	Y = -10.030  mm,	Z = -227.454  mm,
	W = 0.000 deg,	P = 30.000 deg,	R = 160.000 deg
};
P[235]{
   GP1:
	UF : 0, UT : 1,		CONFIG : 'N U T, 0, 0, 0',
	X = 1199.853  mm,	Y = -8.586  mm,	Z = -227.754  mm,
	W = 0.000 deg,	P = 30.000 deg,	R = 160.000 deg
};
P[236]{
   GP1:
	UF : 0, UT : 1,		CONFIG : 'N U T, 0, 0, 0',
	X = 1201.204  mm,	Y = -7.143  mm,	Z = -228.054  mm,
	W = 0.000 deg,	P = 30.000 deg,	R = 160.000 deg
};
P[237]{
   GP1:
	UF : 0, UT : 1,		CONFIG : 'N U T, 0, 0, 0',
	X = 1202.555  mm,	Y = -5.699  mm,	Z = -228.355  mm,
	W = 0.000 deg,	P = 30.000 deg,	R = 160.000 deg
};
P[238]{
   GP1:
	UF : 0, UT : 1,		CONFIG : 'N U T, 0, 0, 0',
	X = 1203.907  mm,	Y = -4.256  mm,	Z = -228.655  mm,
	W = 0.000 deg,	P = 30.000 deg,	R = 160.000 deg
};
P[239]{
   GP1:
	UF : 0, UT : 1,		CONFIG : 'N U T, 0, 0, 0',
	X = 1205.258  mm,	Y = -2.812  mm,	Z = -228.955  mm,
	W = 0.000 deg,	P = 30.000 deg,	R = 160.000 deg
};
P[240]{
   GP1:
	UF : 0, UT : 1,		CONFIG : 'N U T, 0, 0, 0',
	X = 1206.609  mm,	Y = -1.369  mm,	Z = -229.256  mm,
	W = 0.000 deg,	P = 30.000 deg,	R = 160.000 deg
};
P[241]{
   GP1:
	UF : 0, UT : 1,		CONFIG : 'N U T, 0, 0, 0',
	X = 1207.961  mm,	Y = 0.075  mm,	Z = -229.556  mm,
	W = 0.000 deg,	P = 30.000 deg,	R = 160.000 deg
};
P[242]{
   GP1:
	UF : 0, UT : 1,		CONFIG : 'N U T, 0, 0, 0',
	X = 1209.312  mm,	Y = 1.519  mm,	Z = -229.856  mm,
	W = 0.000 deg,	P = 30.000 deg,	R = 160.000 deg
};
P[243]{
   GP1:
	UF : 0, UT : 1,		CONFIG : 'N U T, 0, 0, 0',
	X = 1210.663  mm,	Y = 2.962  mm,	Z = -230.157  mm,
	W = 0.000 deg,	P = 30.000 deg,	R = 160.000 deg
};
P[244]{
   GP1:
	UF : 0, UT : 1,		CONFIG : 'N U T, 0, 0, 0',
	X = 1212.015  mm,	Y = 4.406  mm,	Z = -230.457  mm,
	W = 0.000 deg,	P = 30.000 deg,	R = 160.000 deg
};
P[245]{
   GP1:
	UF : 0, UT : 1,		CONFIG : 'N U T, 0, 0, 0',
	X = 1213.366  mm,	Y = 5.849  mm,	Z = -230.757  mm,
	W = 0.000 deg,	P = 30.000 deg,	R = 160.000 deg
};
P[246]{
   GP1:
	UF : 0, UT : 1,		CONFIG : 'N U T, 0, 0, 0',
	X = 1214.717  mm,	Y = 7.293  mm,	Z = -231.057  mm,
	W = 0.000 deg,	P = 30.000 deg,	R = 160.000 deg
};
P[247]{
   GP1:
	UF : 0, UT : 1,		CONFIG : 'N U T, 0, 0, 0',
	X = 1216.069  mm,	Y = 8.736  mm,	Z = -231.358  mm,
	W = 0.000 deg,	P = 30.000 deg,	R = 160.000 deg
};
P[248]{
   GP1:
	UF : 0, UT : 1,		CONFIG : 'N U T, 0, 0, 0',
	X = 1217.420  mm,	Y = 10.180  mm,	Z = -231.658  mm,
	W = 0.000 deg,	P = 30.000 deg,	R = 160.000 deg
};
P[249]{
   GP1:
	UF : 0, UT : 1,		CONFIG : 'N U T, 0, 0, 0',
	X = 1218.771  mm,	Y = 11.623  mm,	Z = -231.958  mm,
	W = 0.000 deg,	P = 30.000 deg,	R = 160.000 deg
};
P[250]{
   GP1:
	UF : 0, UT : 1,		CONFIG : 'N U T, 0, 0, 0',
	X = 1220.123  mm,	Y = 13.067  mm,	Z = -232.259  mm,
	W = 0.000 deg,	P = 30.000 deg,	R = 160.000 deg
};
P[251]{
   GP1:
	UF : 0, UT : 1,		CONFIG : 'N U T, 0, 0, 0',
	X = 1221.474  mm,	Y = 14.510  mm,	Z = -232.559  mm,
	W = 0.000 deg,	P = 30.000 deg,	R = 160.000 deg
};
P[252]{
   GP1:
	UF : 0, UT : 1,		CONFIG : 'N U T, 0, 0, 0',
	X = 1222.825  mm,	Y = 15.954  mm,	Z = -232.859  mm,
	W = 0.000 deg,	P = 30.000 deg,	R = 160.000 deg
};
P[253]{
   GP1:
	UF : 0, UT : 1,		CONFIG : 'N U T, 0, 0, 0',
	X = 1224.177  mm,	Y = 17.397  mm,	Z = -233.160  mm,
	W = 0.000 deg,	P = 30.000 deg,	R = 160.000 deg
};
P[254]{
   GP1:
	UF : 0, UT : 1,		CONFIG : 'N U T, 0, 0, 0',
	X = 1225.528  mm,	Y = 18.841  mm,	Z = -233.460  mm,
	W = 0.000 deg,	P = 30.000 deg,	R = 160.331 deg
};
P[255]{
   GP1:
	UF : 0, UT : 1,		CONFIG : 'N U T, 0, 0, 0',
	X = 1226.879  mm,	Y = 20.284  mm,	Z = -233.760  mm,
	W = 0.000 deg,	P = 30.000 deg,	R = 164.720 deg
};
P[256]{
   GP1:
	UF : 0, UT : 1,		CONFIG : 'N U T, 0, 0, 0',
	X = 1228.231  mm,	Y = 21.728  mm,	Z = -234.061  mm,
	W = 0.000 deg,	P = 30.000 deg,	R = 169.110 deg
};
P[257]{
   GP1:
	UF : 0, UT : 1,		CONFIG : 'N U T, 0, 0, 0',
	X = 1229.582  mm,	Y = 23.171  mm,	Z = -234.361  mm,
	W = 0.000 deg,	P = 30.000 deg,	R = 173.499 deg
};
P[258]{
   GP1:
	UF : 0, UT : 1,		CONFIG : 'N U T, 0, 0, 0',
	X = 1230.933  mm,	Y = 24.615  mm,	Z = -234.661  mm,
	W = 0.000 deg,	P = 30.000 deg,	R = 177.889 deg
};
P[259]{
   GP1:
	UF : 0, UT : 1,		CONFIG : 'N U T, 0, 0, 0',
	X = 1232.193  mm,	Y = 25.959  mm,	Z = -234.941  mm,
	W = 0.000 deg,	P = 30.000 deg,	R = -178.052 deg
};
P[260]{
   GP1:
	UF : 0, UT : 1,		CONFIG : 'N U T, 0, 0, 0',
	X = 1232.188  mm,	Y = 26.096  mm,	Z = -234.939  mm,
	W = 0.000 deg,	P = 30.000 deg,	R = -178.052 deg
};
P[261]{
   GP1:
	UF : 0, UT : 1,		CONFIG : 'N U T, 0, 0, 0',
	X = 1232.120  mm,	Y = 28.095  mm,	Z = -234.906  mm,
	W = 0.000 deg,	P = 30.000 deg,	R = -178.052 deg
};
P[262]{
   GP1:
	UF : 0, UT : 1,		CONFIG : 'N U T, 0, 0, 0',
	X = 1232.052  mm,	Y = 30.093  mm,	Z = -234.874  mm,
	W = 0.000 deg,	P = 30.000 deg,	R = -178.052 deg
};
P[263]{
   GP1:
	UF : 0, UT : 1,		CONFIG : 'N U T, 0, 0, 0',
	X = 1231.984  mm,	Y = 32.092  mm,	Z = -234.842  mm,
	W = 0.000 deg,	P = 30.000 deg,	R = -178.052 deg
};
P[264]{
   GP1:
	UF : 0, UT : 1,		CONFIG : 'N U T, 0, 0, 0',
	X = 1231.916  mm,	Y = 34.090  mm,	Z = -234.810  mm,
	W = 0.000 deg,	P = 30.000 deg,	R = -178.052 deg
};
P[265]{
   GP1:
	UF : 0, UT : 1,		CONFIG : 'N U T, 0, 0, 0',
	X = 1231.848  mm,	Y = 36.089  mm,	Z = -234.778  mm,
	W = 0.000 deg,	P = 30.000 deg,	R = -178.052 deg
};
P[266]{
   GP1:
	UF : 0, UT : 1,		CONFIG : 'N U T, 0, 0, 0',
	X = 1231.780  mm,	Y = 38.087  mm,	Z = -234.745  mm,
	W = 0.000 deg,	P = 30.000 deg,	R = -178.052 deg
};
P[267]{
   GP1:
	UF : 0, UT : 1,		CONFIG : 'N U T, 0, 0, 0',
	X = 1231.712  mm,	Y = 40.086  mm,	Z = -234.713  mm,
	W = 0.000 deg,	P = 30.000 deg,	R = -178.052 deg
};
P[268]{
   GP1:
	UF : 0, UT : 1,		CONFIG : 'N U T, 0, 0, 0',
	X = 1231.644  mm,	Y = 42.085  mm,	Z = -234.681  mm,
	W = 0.000 deg,	P = 30.000 deg,	R = -178.052 deg
};
P[269]{
   GP1:
	UF : 0, UT : 1,		CONFIG : 'N U T, 0, 0, 0',
	X = 1231.576  mm,	Y = 44.083  mm,	Z = -234.649  mm,
	W = 0.000 deg,	P = 30.000 deg,	R = -178.052 deg
};
P[270]{
   GP1:
	UF : 0, UT : 1,		CONFIG : 'N U T, 0, 0, 0',
	X = 1231.508  mm,	Y = 46.082  mm,	Z = -234.616  mm,
	W = 0.000 deg,	P = 30.000 deg,	R = -178.052 deg
};
P[271]{
   GP1:
	UF : 0, UT : 1,		CONFIG : 'N U T, 0, 0, 0',
	X = 1231.440  mm,	Y = 48.080  mm,	Z = -234.584  mm,
	W = 0.000 deg,	P = 30.000 deg,	R = -178.052 deg
};
P[272]{
   GP1:
	UF : 0, UT : 1,		CONFIG : 'N U T, 0, 0, 0',
	X = 1231.372  mm,	Y = 50.079  mm,	Z = -234.552  mm,
	W = 0.000 deg,	P = 30.000 deg,	R = -178.052 deg
};
P[273]{
   GP1:
	UF : 0, UT : 1,		CONFIG : 'N U T, 0, 0, 0',
	X = 1231.304  mm,	Y = 52.078  mm,	Z = -234.520  mm,
	W = 0.000 deg,	P = 30.000 deg,	R = -178.052 deg
};
P[274]{
   GP1:
	UF : 0, UT : 1,		CONFIG : 'N U T, 0, 0, 0',
	X = 1231.236  mm,	Y = 54.076  mm,	Z = -234.488  mm,
	W = 0.000 deg,	P = 30.000 deg,	R = -178.052 deg
};
P[275]{
   GP1:
	UF : 0, UT : 1,		CONFIG : 'N U T, 0, 0, 0',
	X = 1231.168  mm,	Y = 56.075  mm,	Z = -234.455  mm,
	W = 0.000 deg,	P = 30.000 deg,	R = -178.052 deg
};
P[276]{
   GP1:
	UF : 0, UT : 1,		CONFIG : 'N U T, 0, 0, 0',
	X = 1231.100  mm,	Y = 58.073  mm,	Z = -234.423  mm,
	W = 0.000 deg,	P = 30.000 deg,	R = -178.052 deg
};
P[277]{
   GP1:
	UF : 0, UT : 1,		CONFIG : 'N U T, 0, 0, 0',
	X = 1231.032  mm,	Y = 60.072  mm,	Z = -234.391  mm,
	W = 0.000 deg,	P = 30.000 deg,	R = -178.052 deg
};
P[278]{
   GP1:
	UF : 0, UT : 1,		CONFIG : 'N U T, 0, 0, 0',
	X = 1230.964  mm,	Y = 62.071  mm,	Z = -234.359  mm,
	W = 0.000 deg,	P = 30.000 deg,	R = -178.052 deg
};
P[279]{
   GP1:
	UF : 0, UT : 1,		CONFIG : 'N U T, 0, 0, 0',
	X = 1230.896  mm,	Y = 64.069  mm,	Z = -234.326  mm,
	W = 0.000 deg,	P = 30.000 deg,	R = -178.052 deg
};
P[280]{
   GP1:
	UF : 0, UT : 1,		CONFIG : 'N U T, 0, 0, 0',
	X = 1230.828  mm,	Y = 66.068  mm,	Z = -234.294  mm,
	W = 0.000 deg,	P = 30.000 deg,	R = -178.052 deg
};
P[281]{
   GP1:
	UF : 0, UT : 1,		CONFIG : 'N U T, 0, 0, 0',
	X = 1230.760  mm,	Y = 68.066  mm,	Z = -234.262  mm,
	W = 0.000 deg,	P = 30.000 deg,	R = -178.052 deg
};
P[282]{
   GP1:
	UF : 0, UT : 1,		CONFIG : 'N U T, 0, 0, 0',
	X = 1230.692  mm,	Y = 70.065  mm,	Z = -234.230  mm,
	W = 0.000 deg,	P = 30.000 deg,	R = -178.052 deg
};
P[283]{
   GP1:
	UF : 0, UT : 1,		CONFIG : 'N U T, 0, 0, 0',
	X = 1230.624  mm,	Y = 72.063  mm,	Z = -234.198  mm,
	W = 0.000 deg,	P = 30.000 deg,	R = -178.052 deg
};
P[284]{
   GP1:
	UF : 0, UT : 1,		CONFIG : 'N U T, 0, 0, 0',
	X = 1230.556  mm,	Y = 74.062  mm,	Z = -234.165  mm,
	W = 0.000 deg,	P = 30.000 deg,	R = -174.195 deg
};
P[285]{
   GP1:
	UF : 0, UT : 1,		CONFIG : 'N U T, 0, 0, 0',
	X = 1230.488  mm,	Y = 76.061  mm,	Z = -234.133  mm,
	W = 0.000 deg,	P = 30.000 deg,	R = -170.585 deg
};
P[286]{
   GP1:
	UF : 0, UT : 1,		CONFIG : 'N U T, 0, 0, 0',
	X = 1230.420  mm,	Y = 78.059  mm,	Z = -234.101  mm,
	W = 0.000 deg,	P = 30.000 deg,	R = -166.974 deg
};
P[287]{
   GP1:
	UF : 0, UT : 1,		CONFIG : 'N U T, 0, 0, 0',
	X = 1230.352  mm,	Y = 80.058  mm,	Z = -234.069  mm,
	W = 0.000 deg,	P = 30.000 deg,	R = -163.364 deg
};
P[288]{
   GP1:
	UF : 0, UT : 1,		CONFIG : 'N U T, 0, 0, 0',
	X = 1230.284  mm,	Y = 82.056  mm,	Z = -234.036  mm,
	W = 0.000 deg,	P = 30.000 deg,	R = -160.000 deg
};
P[289]{
   GP1:
	UF : 0, UT : 1,		CONFIG : 'N U T, 0, 0, 0',
	X = 1230.257  mm,	Y = 82.873  mm,	Z = -234.023  mm,
	W = 0.000 deg,	P = 30.000 deg,	R = -160.000 deg
};
P[290]{
   GP1:
	UF : 0, UT : 1,		CONFIG : 'N U T, 0, 0, 0',
	X = 1229.443  mm,	Y = 83.711  mm,	Z = -233.836  mm,
	W = 0.000 deg,	P = 30.000 deg,	R = -160.000 deg
};
P[291]{
   GP1:
	UF : 0, UT : 1,		CONFIG : 'N U T, 0, 0, 0',
	X = 1228.067  mm,	Y = 85.128  mm,	Z = -233.520  mm,
	W = 0.000 deg,	P = 30.000 deg,	R = -160.000 deg
};
P[292]{
   GP1:
	UF : 0, UT : 1,		CONFIG : 'N U T, 0, 0, 0',
	X = 1226.692  mm,	Y = 86.545  mm,	Z = -233.203  mm,
	W = 0.000 deg,	P = 30.000 deg,	R = -160.000 deg
};
P[293]{
   GP1:
	UF : 0, UT : 1,		CONFIG : 'N U T, 0, 0, 0',
	X = 1225.316  mm,	Y = 87.961  mm,	Z = -232.887  mm,
	W = 0.000 deg,	P = 30.000 deg,	R = -160.000 deg
};
P[294]{
   GP1:
	UF : 0, UT : 1,		CONFIG : 'N U T, 0, 0, 0',
	X = 1223.940  mm,	Y = 89.378  mm,	Z = -232.571  mm,
	W = 0.000 deg,	P = 30.000 deg,	R = -160.000 deg
};
P[295]{
   GP1:
	UF : 0, UT : 1,		CONFIG : 'N U T, 0, 0, 0',
	X = 1222.565  mm,	Y = 90.795  mm,	Z = -232.254  mm,
	W = 0.000 deg,	P = 30.000 deg,	R = -160.000 deg
};
P[296]{
   GP1:
	UF : 0, UT : 1,		CONFIG : 'N U T, 0, 0, 0',
	X = 1221.189  mm,	Y = 92.212  mm,	Z = -231.938  mm,
	W = 0.000 deg,	P = 30.000 deg,	R = -160.000 deg
};
P[297]{
   GP1:
	UF : 0, UT : 1,		CONFIG : 'N U T, 0, 0, 0',
	X = 1219.814  mm,	Y = 93.629  mm,	Z = -231.621  mm,
	W = 0.000 deg,	P = 30.000 deg,	R = -160.000 deg
};
P[298]{
   GP1:
	UF : 0, UT : 1,		CONFIG : 'N U T, 0, 0, 0',
	X = 1218.438  mm,	Y = 95.046  mm,	Z = -231.305  mm,
	W = 0.000 deg,	P = 30.000 deg,	R = -160.000 deg
};
P[299]{
   GP1:
	UF : 0, UT : 1,		CONFIG : 'N U T, 0, 0, 0',
	X = 1217.062  mm,	Y = 96.463  mm,	Z = -230.989  mm,
	W = 0.000 deg,	P = 30.000 deg,	R = -160.000 deg
};
P[300]{
   GP1:
	UF : 0, UT : 1,		CONFIG : 'N U T, 0, 0, 0',
	X = 1215.687  mm,	Y = 97.879  mm,	Z = -230.672  mm,
	W = 0.000 deg,	P = 30.000 deg,	R = -160.000 deg
};
P[301]{
   GP1:
	UF : 0, UT : 1,		CONFIG : 'N U T, 0, 0, 0',
	X = 1214.311  mm,	Y = 99.296  mm,	Z = -230.356  mm,
	W = 0.000 deg,	P = 30.000 deg,	R = -160.000 deg
};
P[302]{
   GP1:
	UF : 0, UT : 1,		CONFIG : 'N U T, 0, 0, 0',
	X = 1212.935  mm,	Y = 100.713  mm,	Z = -230.039  mm,
	W = 0.000 deg,	P = 30.000 deg,	R = -160.000 deg
};
P[303]{
   GP1:
	UF : 0, UT : 1,		CONFIG : 'N U T, 0, 0, 0',
	X = 1211.560  mm,	Y = 102.130  mm,	Z = -229.723  mm,
	W = 0.000 deg,	P = 30.000 deg,	R = -160.000 deg
};
P[304]{
   GP1:
	UF : 0, UT : 1,		CONFIG : 'N U T, 0, 0, 0',
	X = 1210.184  mm,	Y = 103.547  mm,	Z = -229.407  mm,
	W = 0.000 deg,	P = 30.000 deg,	R = -160.000 deg
};
P[305]{
   GP1:
	UF : 0, UT : 1,		CONFIG : 'N U T, 0, 0, 0',
	X = 1208.808  mm,	Y = 104.964  mm,	Z = -229.090  mm,
	W = 0.000 deg,	P = 30.000 deg,	R = -160.000 deg
};
P[306]{
   GP1:
	UF : 0, UT : 1,		CONFIG : 'N U T, 0, 0, 0',
	X = 1207.433  mm,	Y = 106.381  mm,	Z = -228.774  mm,
	W = 0.000 deg,	P = 30.000 deg,	R = -160.000 deg
};
P[307]{
   GP1:
	UF : 0, UT : 1,		CONFIG : 'N U T, 0, 0, 0',
	X = 1206.057  mm,	Y = 107.797  mm,	Z = -228.458  mm,
	W = 0.000 deg,	P = 30.000 deg,	R = -160.000 deg
};
P[308]{
   GP1:
	UF : 0, UT : 1,		CONFIG : 'N U T, 0, 0, 0',
	X = 1204.681  mm,	Y = 109.214  mm,	Z = -228.141  mm,
	W = 0.000 deg,	P = 30.000 deg,	R = -160.000 deg
};
P[309]{
   GP1:
	UF : 0, UT : 1,		CONFIG : 'N U T, 0, 0, 0',
	X = 1203.306  mm,	Y = 110.631  mm,	Z = -227.825  mm,
	W = 0.000 deg,	P = 30.000 deg,	R = -160.000 deg
};
P[310]{
   GP1:
	UF : 0, UT : 1,		CONFIG : 'N U T, 0, 0, 0',
	X = 1201.930  mm,	Y = 112.048  mm,	Z = -227.508  mm,
	W = 0.000 deg,	P = 30.000 deg,	R = -160.000 deg
};
P[311]{
   GP1:
	UF : 0, UT : 1,		CONFIG : 'N U T, 0, 0, 0',
	X = 1200.554  mm,	Y = 113.465  mm,	Z = -227.192  mm,
	W = 0.000 deg,	P = 30.000 deg,	R = -160.000 deg
};
P[312]{
   GP1:
	UF : 0, UT : 1,		CONFIG : 'N U T, 0, 0, 0',
	X = 1199.179  mm,	Y = 114.882  mm,	Z = -226.876  mm,
	W = 0.000 deg,	P = 30.000 deg,	R = -166.547 deg
};
P[313]{
   GP1:
	UF : 0, UT : 1,		CONFIG : 'N U T, 0, 0, 0',
	X = 1197.803  mm,	Y = 116.299  mm,	Z = -226.559  mm,
	W = 0.000 deg,	P = 30.000 deg,	R = -170.662 deg
};
P[314]{
   GP1:
	UF : 0, UT : 1,		CONFIG : 'N U T, 0, 0, 0',
	X = 1196.427  mm,	Y = 117.715  mm,	Z = -226.243  mm,
	W = 0.000 deg,	P = 30.000 deg,	R = -174.776 deg
};
P[315]{
   GP1:
	UF : 0, UT : 1,		CONFIG : 'N U T, 0, 0, 0',
	X = 1195.052  mm,	Y = 119.132  mm,	Z = -225.926  mm,
	W = 0.000 deg,	P = 30.000 deg,	R = -178.890 deg
};
P[316]{
   GP1:
	UF : 0, UT : 1,		CONFIG : 'N U T, 0, 0, 0',
	X = 1193.972  mm,	Y = 120.244  mm,	Z = -225.678  mm,
	W = 0.000 deg,	P = 30.000 deg,	R = 179.429 deg
};
P[317]{
   GP1:
	UF : 0, UT : 1,		CONFIG : 'N U T, 0, 0, 0',
	X = 1193.976  mm,	Y = 120.675  mm,	Z = -225.672  mm,
	W = 0.000 deg,	P = 30.000 deg,	R = 179.429 deg
};
P[318]{
   GP1:
	UF : 0, UT : 1,		CONFIG : 'N U T, 0, 0, 0',
	X = 1193.996  mm,	Y = 122.674  mm,	Z = -225.646  mm,
	W = 0.000 deg,	P = 30.000 deg,	R = 179.429 deg
};
P[319]{
   GP1:
	UF : 0, UT : 1,		CONFIG : 'N U T, 0, 0, 0',
	X = 1194.016  mm,	Y = 124.674  mm,	Z = -225.620  mm,
	W = 0.000 deg,	P = 30.000 deg,	R = 179.429 deg
};
P[320]{
   GP1:
	UF : 0, UT : 1,		CONFIG : 'N U T, 0, 0, 0',
	X = 1194.036  mm,	Y = 126.674  mm,	Z = -225.594  mm,
	W = 0.000 deg,	P = 30.000 deg,	R = 179.429 deg
};
P[321]{
   GP1:
	UF : 0, UT : 1,		CONFIG : 'N U T, 0, 0, 0',
	X = 1194.056  mm,	Y = 128.673  mm,	Z = -225.567  mm,
	W = 0.000 deg,	P = 30.000 deg,	R = 179.429 deg
};
P[322]{
   GP1:
	UF : 0, UT : 1,		CONFIG : 'N U T, 0, 0, 0',
	X = 1194.076  mm,	Y = 130.673  mm,	Z = -225.541  mm,
	W = 0.000 deg,	P = 30.000 deg,	R = 179.429 deg
};
P[323]{
   GP1:
	UF : 0, UT : 1,		CONFIG : 'N U T, 0, 0, 0',
	X = 1194.096  mm,	Y = 132.673  mm,	Z = -225.515  mm,
	W = 0.000 deg,	P = 30.000 deg,	R = 179.429 deg
};
P[324]{
   GP1:
	UF : 0, UT : 1,		CONFIG : 'N U T, 0, 0, 0',
	X = 1194.116  mm,	Y = 134.673  mm,	Z = -225.489  mm,
	W = 0.000 deg,	P = 30.000 deg,	R = 179.429 deg
};
P[325]{
   GP1:
	UF : 0, UT : 1,		CONFIG : 'N U T, 0, 0, 0',
	X = 1194.136  mm,	Y = 136.672  mm,	Z = -225.462  mm,
	W = 0.000 deg,	P = 30.000 deg,	R = 179.429 deg
};
P[326]{
   GP1:
	UF : 0, UT : 1,		CONFIG : 'N U T, 0, 0, 0',
	X = 1194.156  mm,	Y = 138.672  mm,	Z = -225.436  mm,
	W = 0.000 deg,	P = 30.000 deg,	R = 179.429 deg
};
P[327]{
   GP1:
	UF : 0, UT : 1,		CONFIG : 'N U T, 0, 0, 0',
	X = 1194.176  mm,	Y = 140.672  mm,	Z = -225.410  mm,
	W = 0.000 deg,	P = 30.000 deg,	R = 179.429 deg
};
P[328]{
   GP1:
	UF : 0, UT : 1,		CONFIG : 'N U T, 0, 0, 0',
	X = 1194.196  mm,	Y = 142.672  mm,	Z = -225.384  mm,
	W = 0.000 deg,	P = 30.000 deg,	R = 179.429 deg
};
P[329]{
   GP1:
	UF : 0, UT : 1,		CONFIG : 'N U T, 0, 0, 0',
	X = 1194.215  mm,	Y = 144.671  mm,	Z = -225.357  mm,
	W = 0.000 deg,	P = 30.000 deg,	R = 179.429 deg
};
P[330]{
   GP1:
	UF : 0, UT : 1,		CONFIG : 'N U T, 0, 0, 0',
	X = 1194.235  mm,	Y = 146.671  mm,	Z = -225.331  mm,
	W = 0.000 deg,	P = 30.000 deg,	R = 179.429 deg
};
P[331]{
   GP1:
	UF : 0, UT : 1,		CONFIG : 'N U T, 0, 0, 0',
	X = 1194.255  mm,	Y = 148.671  mm,	Z = -225.305  mm,
	W = 0.000 deg,	P = 30.000 deg,	R = 179.429 deg
};
P[332]{
   GP1:
	UF : 0, UT : 1,		CONFIG : 'N U T, 0, 0, 0',
	X = 1194.275  mm,	Y = 150.670  mm,	Z = -225.278  mm,
	W = 0.000 deg,	P = 30.000 deg,	R = 179.429 deg
};
P[333]{
   GP1:
	UF : 0, UT : 1,		CONFIG : 'N U T, 0, 0, 0',
	X = 1194.295  mm,	Y = 152.670  mm,	Z = -225.252  mm,
	W = 0.000 deg,	P = 30.000 deg,	R = 179.429 deg
};
P[334]{
   GP1:
	UF : 0, UT : 1,		CONFIG : 'N U T, 0, 0, 0',
	X = 1194.315  mm,	Y = 154.670  mm,	Z = -225.226  mm,
	W = 0.000 deg,	P = 30.000 deg,	R = 179.429 deg
};
P[335]{
   GP1:
	UF : 0, UT : 1,		CONFIG : 'N U T, 0, 0, 0',
	X = 1194.335  mm,	Y = 156.670  mm,	Z = -225.200  mm,
	W = 0.000 deg,	P = 30.000 deg,	R = 179.429 deg
};
P[336]{
   GP1:
	UF : 0, UT : 1,		CONFIG : 'N U T, 0, 0, 0',
	X = 1194.355  mm,	Y = 158.669  mm,	Z = -225.173  mm,
	W = 0.000 deg,	P = 30.000 deg,	R = 179.429 deg
};
P[337]{
   GP1:
	UF : 0, UT : 1,		CONFIG : 'N U T, 0, 0, 0',
	X = 1194.375  mm,	Y = 160.669  mm,	Z = -225.147  mm,
	W = 0.000 deg,	P = 30.000 deg,	R = 179.429 deg
};
P[338]{
   GP1:
	UF : 0, UT : 1,		CONFIG : 'N U T, 0, 0, 0',
	X = 1194.395  mm,	Y = 162.669  mm,	Z = -225.121  mm,
	W = 0.000 deg,	P = 30.000 deg,	R = 179.429 deg
};
P[339]{
   GP1:
	UF : 0, UT : 1,		CONFIG : 'N U T, 0, 0, 0',
	X = 1194.415  mm,	Y = 164.669  mm,	Z = -225.095  mm,
	W = 0.000 deg,	P = 30.000 deg,	R = 179.429 deg
};
P[340]{
   GP1:
	UF : 0, UT : 1,		CONFIG : 'N U T, 0, 0, 0',
	X = 1194.435  mm,	Y = 166.668  mm,	Z = -225.068  mm,
	W = 0.000 deg,	P = 30.000 deg,	R = 179.429 deg
};
P[341]{
   GP1:
	UF : 0, UT : 1,		CONFIG : 'N U T, 0, 0, 0',
	X = 1194.455  mm,	Y = 168.668  mm,	Z = -225.042  mm,
	W = 0.000 deg,	P = 30.000 deg,	R = 178.593 deg
};
P[342]{
   GP1:
	UF : 0, UT : 1,		CONFIG : 'N U T, 0, 0, 0',
	X = 1194.475  mm,	Y = 170.668  mm,	Z = -225.016  mm,
	W = 0.000 deg,	P = 30.000 deg,	R = 174.707 deg
};
P[343]{
   GP1:
	UF : 0, UT : 1,		CONFIG : 'N U T, 0, 0, 0',
	X = 1194.495  mm,	Y = 172.667  mm,	Z = -224.989  mm,
	W = 0.000 deg,	P = 30.000 deg,	R = 170.822 deg
};
P[344]{
   GP1:
	UF : 0, UT : 1,		CONFIG : 'N U T, 0, 0, 0',
	X = 1194.514  mm,	Y = 174.667  mm,	Z = -224.963  mm,
	W = 0.000 deg,	P = 30.000 deg,	R = 166.936 deg
};
P[345]{
   GP1:
	UF : 0, UT : 1,		CONFIG : 'N U T, 0, 0, 0',
	X = 1194.534  mm,	Y = 176.667  mm,	Z = -224.937  mm,
	W = 0.000 deg,	P = 30.000 deg,	R = 163.050 deg
};
P[346]{
   GP1:
	UF : 0, UT : 1,		CONFIG : 'N U T, 0, 0, 0',
	X = 1194.552  mm,	Y = 178.418  mm,	Z = -224.914  mm,
	W = 0.000 deg,	P = 30.000 deg,	R = 160.000 deg
};
P[347]{
   GP1:
	UF : 0, UT : 1,		CONFIG : 'N U T, 0, 0, 0',
	X = 1194.720  mm,	Y = 178.597  mm,	Z = -224.954  mm,
	W = 0.000 deg,	P = 30.000 deg,	R = 160.000 deg
};
P[348]{
   GP1:
	UF : 0, UT : 1,		CONFIG : 'N U T, 0, 0, 0',
	X = 1196.074  mm,	Y = 180.033  mm,	Z = -225.276  mm,
	W = 0.000 deg,	P = 30.000 deg,	R = 160.000 deg
};
P[349]{
   GP1:
	UF : 0, UT : 1,		CONFIG : 'N U T, 0, 0, 0',
	X = 1197.427  mm,	Y = 181.470  mm,	Z = -225.599  mm,
	W = 0.000 deg,	P = 30.000 deg,	R = 160.000 deg
};
P[350]{
   GP1:
	UF : 0, UT : 1,		CONFIG : 'N U T, 0, 0, 0',
	X = 1198.781  mm,	Y = 182.907  mm,	Z = -225.921  mm,
	W = 0.000 deg,	P = 30.000 deg,	R = 160.000 deg
};
P[351]{
   GP1:
	UF : 0, UT : 1,		CONFIG : 'N U T, 0, 0, 0',
	X = 1200.134  mm,	Y = 184.343  mm,	Z = -226.243  mm,
	W = 0.000 deg,	P = 30.000 deg,	R = 160.000 deg
};
P[352]{
   GP1:
	UF : 0, UT : 1,		CONFIG : 'N U T, 0, 0, 0',
	X = 1201.488  mm,	Y = 185.780  mm,	Z = -226.565  mm,
	W = 0.000 deg,	P = 30.000 deg,	R = 160.000 deg
};
P[353]{
   GP1:
	UF : 0, UT : 1,		CONFIG : 'N U T, 0, 0, 0',
	X = 1202.841  mm,	Y = 187.217  mm,	Z = -226.888  mm,
	W = 0.000 deg,	P = 30.000 deg,	R = 160.000 deg
};
P[354]{
   GP1:
	UF : 0, UT : 1,		CONFIG : 'N U T, 0, 0, 0',
	X = 1204.195  mm,	Y = 188.653  mm,	Z = -227.210  mm,
	W = 0.000 deg,	P = 30.000 deg,	R = 160.000 deg
};
P[355]{
   GP1:
	UF : 0, UT : 1,		CONFIG : 'N U T, 0, 0, 0',
	X = 1205.549  mm,	Y = 190.090  mm,	Z = -227.532  mm,
	W = 0.000 deg,	P = 30.000 deg,	R = 160.000 deg
};
P[356]{
   GP1:
	UF : 0, UT : 1,		CONFIG : 'N U T, 0, 0, 0',
	X = 1206.902  mm,	Y = 191.527  mm,	Z = -227.854  mm,
	W = 0.000 deg,	P = 30.000 deg,	R = 160.000 deg
};
P[357]{
   GP1:
	UF : 0, UT : 1,		CONFIG : 'N U T, 0, 0, 0',
	X = 1208.256  mm,	Y = 192.964  mm,	Z = -228.177  mm,
	W = 0.000 deg,	P = 30.000 deg,	R = 160.000 deg
};
P[358]{
   GP1:
	UF : 0, UT : 1,		CONFIG : 'N U T, 0, 0, 0',
	X = 1209.609  mm,	Y = 194.400  mm,	Z = -228.499  mm,
	W = 0.000 deg,	P = 30.000 deg,	R = 160.000 deg
};
P[359]{
   GP1:
	UF : 0, UT : 1,		CONFIG : 'N U T, 0, 0, 0',
	X = 1210.963  mm,	Y = 195.837  mm,	Z = -228.821  mm,
	W = 0.000 deg,	P = 30.000 deg,	R = 160.000 deg
};
P[360]{
   GP1:
	UF : 0, UT : 1,		CONFIG : 'N U T, 0, 0, 0',
	X = 1212.316  mm,	Y = 197.274  mm,	Z = -229.143  mm,
	W = 0.000 deg,	P = 30.000 deg,	R = 160.000 deg
};
P[361]{
   GP1:
	UF : 0, UT : 1,		CONFIG : 'N U T, 0, 0, 0',
	X = 1213.670  mm,	Y = 198.710  mm,	Z = -229.466  mm,
	W = 0.000 deg,	P = 30.000 deg,	R = 160.000 deg
};
P[362]{
   GP1:
	UF : 0, UT : 1,		CONFIG : 'N U T, 0, 0, 0',
	X = 1215.023  mm,	Y = 200.147  mm,	Z = -229.788  mm,
	W = 0.000 deg,	P = 30.000 deg,	R = 160.000 deg
};
P[363]{
   GP1:
	UF : 0, UT : 1,		CONFIG : 'N U T, 0, 0, 0',
	X = 1216.377  mm,	Y = 201.584  mm,	Z = -230.110  mm,
	W = 0.000 deg,	P = 30.000 deg,	R = 160.000 deg
};
P[364]{
   GP1:
	UF : 0, UT : 1,		CONFIG : 'N U T, 0, 0, 0',
	X = 1217.730  mm,	Y = 203.020  mm,	Z = -230.432  mm,
	W = 0.000 deg,	P = 30.000 deg,	R = 160.000 deg
};
P[365]{
   GP1:
	UF : 0, UT : 1,		CONFIG : 'N U T, 0, 0, 0',
	X = 1219.084  mm,	Y = 204.457  mm,	Z = -230.755  mm,
	W = 0.000 deg,	P = 30.000 deg,	R = 160.000 deg
};
P[366]{
   GP1:
	UF : 0, UT : 1,		CONFIG : 'N U T, 0, 0, 0',
	X = 1220.437  mm,	Y = 205.894  mm,	Z = -231.077  mm,
	W = 0.000 deg,	P = 30.000 deg,	R = 160.000 deg
};
P[367]{
   GP1:
	UF : 0, UT : 1,		CONFIG : 'N U T, 0, 0, 0',
	X = 1221.791  mm,	Y = 207.330  mm,	Z = -231.399  mm,
	W = 0.000 deg,	P = 30.000 deg,	R = 160.000 deg
};
P[368]{
   GP1:
	UF : 0, UT : 1,		CONFIG : 'N U T, 0, 0, 0',
	X = 1223.145  mm,	Y = 208.767  mm,	Z = -231.721  mm,
	W = 0.000 deg,	P = 30.000 deg,	R = 164.334 deg
};
P[369]{
   GP1:
	UF : 0, UT : 1,		CONFIG : 'N U T, 0, 0, 0',
	X = 1224.498  mm,	Y = 210.204  mm,	Z = -232.044  mm,
	W = 0.000 deg,	P = 30.000 deg,	R = 168.188 deg
};
P[370]{
   GP1:
	UF : 0, UT : 1,		CONFIG : 'N U T, 0, 0, 0',
	X = 1225.852  mm,	Y = 211.641  mm,	Z = -232.366  mm,
	W = 0.000 deg,	P = 30.000 deg,	R = 172.043 deg
};
P[371]{
   GP1:
	UF : 0, UT : 1,		CONFIG : 'N U T, 0, 0, 0',
	X = 1227.205  mm,	Y = 213.077  mm,	Z = -232.688  mm,
	W = 0.000 deg,	P = 30.000 deg,	R = 175.897 deg
};
P[372]{
   GP1:
	UF : 0, UT : 1,		CONFIG : 'N U T, 0, 0, 0',
	X = 1228.559  mm,	Y = 214.514  mm,	Z = -233.010  mm,
	W = 0.000 deg,	P = 30.000 deg,	R = 179.272 deg
};
P[373]{
   GP1:
	UF : 0, UT : 1,		CONFIG : 'N U T, 0, 0, 0',
	X = 1229.346  mm,	Y = 215.349  mm,	Z = -233.198  mm,
	W = 0.000 deg,	P = 30.000 deg,	R = 179.272 deg
};
P[374]{
   GP1:
	UF : 0, UT : 1,		CONFIG : 'N U T, 0, 0, 0',
	X = 1229.356  mm,	Y = 216.186  mm,	Z = -233.194  mm,
	W = 0.000 deg,	P = 30.000 deg,	R = 179.272 deg
};
P[375]{
   GP1:
	UF : 0, UT : 1,		CONFIG : 'N U T, 0, 0, 0',
	X = 1229.382  mm,	Y = 218.186  mm,	Z = -233.184  mm,
	W = 0.000 deg,	P = 30.000 deg,	R = 179.272 deg
};
P[376]{
   GP1:
	UF : 0, UT : 1,		CONFIG : 'N U T, 0, 0, 0',
	X = 1229.407  mm,	Y = 220.186  mm,	Z = -233.175  mm,
	W = 0.000 deg,	P = 30.000 deg,	R = 179.272 deg
};
P[377]{
   GP1:
	UF : 0, UT : 1,		CONFIG : 'N U T, 0, 0, 0',
	X = 1229.422  mm,	Y = 221.349  mm,	Z = -233.169  mm,
	W = 0.000 deg,	P = 30.000 deg,	R = 179.272 deg
};
/END
